KUKA KRL program: f1_Kuka_APT220T02S20.SRC

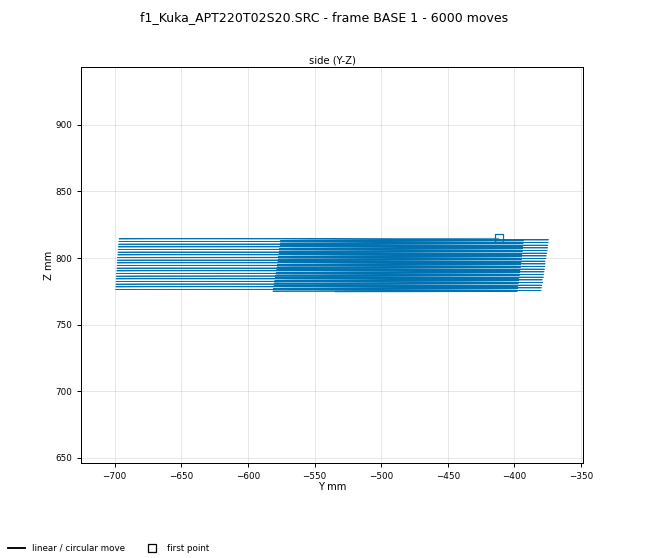
[picture p0: tool path of f1_Kuka_APT220T02S20.SRC in frame BASE 1, 6000 of 6001 moves have a stored position in this frame; points joined in program order, loops and branches not executed]
&ACCESS RVP
&REL 2
&PARAM TEMPLATE = C:\KRC\Roboter\Template\vorgabe
&PARAM EDITMASK = *
DEF f1_Kuka_APT220T02S20()


;FOLD INI;%{PE}%V3.2.0,%MKUKATPBASIS,%CINIT,%VCOMMON,%P
  ;FOLD BAS INI;%{E}%V3.2.0,%MKUKATPBASIS,%CINIT,%VINIT,%P
    GLOBAL INTERRUPT DECL 3 WHEN $STOPMESS==TRUE DO IR_STOPM ( )
    INTERRUPT ON 3
    BAS (#INITMOV,0 )
  ;ENDFOLD (BAS INI)
  ;FOLD USER INI;%{E}%V3.2.0,%MKUKATPUSER,%CINIT,%VINIT,%P
    ;Make your modifications here
  ;ENDFOLD (USER INI)
;ENDFOLD (INI)


;*** Make Null PTP Move
  PTP $pos_act

;*** Auto Load The Correct TOOL Data
  $tool=tool_data[2]

;*** Auto Load The Correct BASE Data
  $base=base_data[1]

  $ADVANCE = 5

;*** Restate Last Velocity
MMPM(30000.0)
SetRPM(8000)
LIN {X 0.104,Y -411.815,Z 814.863,A 0.000,B 0.000,C 90.000,E1 11.243} C_DIS
LIN {X -0.028,Y -415.979,Z 814.849,A 0.000,B 0.000,C 90.000,E1 8.859} C_DIS
LIN {X -0.170,Y -419.674,Z 814.838,A 0.000,B 0.000,C 90.000,E1 6.834} C_DIS
LIN {X 0.068,Y -422.792,Z 814.828,A 0.000,B 0.000,C 90.000,E1 5.106} C_DIS
LIN {X 0.041,Y -427.269,Z 814.815,A 0.000,B 0.000,C 90.000,E1 2.751} C_DIS
LIN {X 0.164,Y -433.422,Z 814.799,A 0.000,B 0.000,C 90.000,E1 359.771} C_DIS
LIN {X -0.033,Y -438.556,Z 814.786,A 0.000,B 0.000,C 90.000,E1 357.478} C_DIS
LIN {X 0.129,Y -442.521,Z 814.777,A 0.000,B 0.000,C 90.000,E1 355.812} C_DIS
LIN {X 0.097,Y -447.330,Z 814.766,A 0.000,B 0.000,C 90.000,E1 353.856} C_DIS
LIN {X 0.027,Y -451.496,Z 814.757,A 0.000,B 0.000,C 90.000,E1 352.243} C_DIS
LIN {X -0.123,Y -454.846,Z 814.750,A 0.000,B 0.000,C 90.000,E1 350.971} C_DIS
LIN {X -0.144,Y -456.848,Z 814.746,A 0.000,B 0.000,C 90.000,E1 350.330} C_DIS
LIN {X 0.078,Y -458.176,Z 814.744,A 0.000,B 0.000,C 90.000,E1 349.982} C_DIS
LIN {X 0.076,Y -460.220,Z 814.742,A 0.000,B 0.000,C 90.000,E1 349.634} C_DIS
LIN {X 0.046,Y -461.513,Z 814.741,A 0.000,B 0.000,C 90.000,E1 349.398} C_DIS
LIN {X 0.102,Y -464.808,Z 814.739,A 0.000,B 0.000,C 90.000,E1 348.993} C_DIS
LIN {X -0.030,Y -469.453,Z 814.737,A 0.000,B 0.000,C 90.000,E1 348.578} C_DIS
LIN {X 0.114,Y -476.009,Z 814.734,A 0.000,B 0.000,C 90.000,E1 348.049} C_DIS
LIN {X 0.121,Y -489.154,Z 814.729,A 0.000,B 0.000,C 90.000,E1 347.173} C_DIS
LIN {X -0.029,Y -500.125,Z 814.725,A 0.000,B 0.000,C 90.000,E1 346.464} C_DIS
LIN {X 0.244,Y -511.204,Z 814.721,A 0.000,B 0.000,C 90.000,E1 345.700} C_DIS
LIN {X 0.051,Y -523.694,Z 814.716,A 0.000,B 0.000,C 90.000,E1 344.866} C_DIS
LIN {X 0.230,Y -535.945,Z 814.711,A 0.000,B 0.000,C 90.000,E1 343.976} C_DIS
LIN {X 0.109,Y -546.247,Z 814.707,A 0.000,B 0.000,C 90.000,E1 343.196} C_DIS
LIN {X 0.238,Y -553.395,Z 814.703,A 0.000,B 0.000,C 90.000,E1 342.598} C_DIS
LIN {X 0.128,Y -558.933,Z 814.701,A 0.000,B 0.000,C 90.000,E1 342.127} C_DIS
LIN {X 0.040,Y -565.603,Z 814.697,A 0.000,B 0.000,C 90.000,E1 341.511} C_DIS
LIN {X 0.103,Y -571.834,Z 814.694,A 0.000,B 0.000,C 90.000,E1 340.859} C_DIS
LIN {X 0.161,Y -576.778,Z 814.691,A 0.000,B 0.000,C 90.000,E1 340.315} C_DIS
LIN {X 0.095,Y -582.280,Z 814.687,A 0.000,B 0.000,C 90.000,E1 339.645} C_DIS
LIN {X -0.127,Y -585.378,Z 814.685,A 0.000,B 0.000,C 90.000,E1 339.263} C_DIS
LIN {X 0.313,Y -591.974,Z 814.680,A 0.000,B 0.000,C 90.000,E1 338.284} C_DIS
LIN {X -0.223,Y -597.103,Z 814.675,A 0.000,B 0.000,C 90.000,E1 337.539} C_DIS
LIN {X -0.236,Y -603.578,Z 814.669,A 0.000,B 0.000,C 90.000,E1 336.485} C_DIS
LIN {X 0.161,Y -607.408,Z 814.666,A 0.000,B 0.000,C 90.000,E1 335.793} C_DIS
LIN {X -0.289,Y -614.208,Z 814.659,A 0.000,B 0.000,C 90.000,E1 334.665} C_DIS
LIN {X 0.202,Y -617.825,Z 814.656,A 0.000,B 0.000,C 90.000,E1 333.973} C_DIS
LIN {X 0.166,Y -624.634,Z 814.648,A 0.000,B 0.000,C 90.000,E1 332.692} C_DIS
LIN {X -0.052,Y -629.035,Z 814.643,A 0.000,B 0.000,C 90.000,E1 331.820} C_DIS
LIN {X 0.073,Y -634.391,Z 814.637,A 0.000,B 0.000,C 90.000,E1 330.667} C_DIS
LIN {X 0.046,Y -640.111,Z 814.630,A 0.000,B 0.000,C 90.000,E1 329.410} C_DIS
LIN {X 0.048,Y -644.293,Z 814.625,A 0.000,B 0.000,C 90.000,E1 328.408} C_DIS
LIN {X -0.026,Y -649.093,Z 814.618,A 0.000,B 0.000,C 90.000,E1 327.168} C_DIS
LIN {X 0.087,Y -652.631,Z 814.612,A 0.000,B 0.000,C 90.000,E1 326.167} C_DIS
LIN {X 0.063,Y -655.871,Z 814.607,A 0.000,B 0.000,C 90.000,E1 325.182} C_DIS
LIN {X 0.086,Y -658.937,Z 814.601,A 0.000,B 0.000,C 90.000,E1 324.196} C_DIS
LIN {X 0.103,Y -662.514,Z 814.594,A 0.000,B 0.000,C 90.000,E1 322.970} C_DIS
LIN {X 0.181,Y -665.628,Z 814.588,A 0.000,B 0.000,C 90.000,E1 321.743} C_DIS
LIN {X -0.215,Y -668.498,Z 814.581,A 0.000,B 0.000,C 90.000,E1 320.561} C_DIS
LIN {X 0.375,Y -671.116,Z 814.574,A 0.000,B 0.000,C 90.000,E1 319.299} C_DIS
LIN {X 0.046,Y -673.535,Z 814.567,A 0.000,B 0.000,C 90.000,E1 318.119} C_DIS
LIN {X 0.104,Y -674.880,Z 814.563,A 0.000,B 0.000,C 90.000,E1 317.391} C_DIS
LIN {X -0.220,Y -676.865,Z 814.557,A 0.000,B 0.000,C 90.000,E1 316.215} C_DIS
LIN {X -0.118,Y -677.962,Z 814.553,A 0.000,B 0.000,C 90.000,E1 315.486} C_DIS
LIN {X -0.003,Y -678.964,Z 814.549,A 0.000,B 0.000,C 90.000,E1 314.757} C_DIS
LIN {X 0.207,Y -680.520,Z 814.542,A 0.000,B 0.000,C 90.000,E1 313.542} C_DIS
LIN {X -0.397,Y -682.522,Z 814.533,A 0.000,B 0.000,C 90.000,E1 311.919} C_DIS
LIN {X -0.093,Y -683.878,Z 814.526,A 0.000,B 0.000,C 90.000,E1 310.701} C_DIS
LIN {X -0.161,Y -685.334,Z 814.518,A 0.000,B 0.000,C 90.000,E1 309.277} C_DIS
LIN {X -0.256,Y -686.461,Z 814.512,A 0.000,B 0.000,C 90.000,E1 308.096} C_DIS
LIN {X -0.130,Y -687.930,Z 814.502,A 0.000,B 0.000,C 90.000,E1 306.423} C_DIS
LIN {X -0.057,Y -688.887,Z 814.496,A 0.000,B 0.000,C 90.000,E1 305.231} C_DIS
LIN {X 0.031,Y -689.765,Z 814.489,A 0.000,B 0.000,C 90.000,E1 304.040} C_DIS
LIN {X -0.394,Y -690.938,Z 814.480,A 0.000,B 0.000,C 90.000,E1 302.418} C_DIS
LIN {X 0.163,Y -692.232,Z 814.471,A 0.000,B 0.000,C 90.000,E1 300.718} C_DIS
LIN {X 0.154,Y -693.018,Z 814.464,A 0.000,B 0.000,C 90.000,E1 299.539} C_DIS
LIN {X 0.048,Y -694.134,Z 814.455,A 0.000,B 0.000,C 90.000,E1 297.897} C_DIS
LIN {X 0.255,Y -695.322,Z 814.446,A 0.000,B 0.000,C 90.000,E1 296.232} C_DIS
LIN {X -0.064,Y -696.432,Z 814.438,A 0.000,B 0.000,C 90.000,E1 294.847} C_DIS
LIN {X -0.184,Y -696.729,Z 814.435,A 0.000,B 0.000,C 90.000,E1 294.387} C_DIS
LIN {X 0.044,Y -696.654,Z 814.433,A 0.000,B 0.000,C 90.000,E1 293.898} C_DIS
LIN {X 0.301,Y -696.552,Z 814.432,A 0.000,B 0.000,C 90.000,E1 293.643} C_DIS
LIN {X -0.083,Y -696.012,Z 814.430,A 0.000,B 0.000,C 90.000,E1 293.439} C_DIS
LIN {X 0.146,Y -694.455,Z 814.428,A 0.000,B 0.000,C 90.000,E1 292.950} C_DIS
LIN {X 0.269,Y -693.767,Z 814.427,A 0.000,B 0.000,C 90.000,E1 292.823} C_DIS
LIN {X 0.124,Y -692.737,Z 814.426,A 0.000,B 0.000,C 90.000,E1 292.717} C_DIS
LIN {X -0.273,Y -690.283,Z 814.425,A 0.000,B 0.000,C 90.000,E1 292.514} C_DIS
LIN {X -0.230,Y -687.459,Z 814.424,A 0.000,B 0.000,C 90.000,E1 292.280} C_DIS
LIN {X 0.023,Y -685.623,Z 814.423,A 0.000,B 0.000,C 90.000,E1 292.153} C_DIS
LIN {X 0.071,Y -681.364,Z 814.422,A 0.000,B 0.000,C 90.000,E1 291.972} C_DIS
LIN {X 0.256,Y -675.989,Z 814.421,A 0.000,B 0.000,C 90.000,E1 291.770} C_DIS
LIN {X 0.101,Y -671.875,Z 814.420,A 0.000,B 0.000,C 90.000,E1 291.663} C_DIS
LIN {X -0.284,Y -662.431,Z 814.420,A 0.000,B 0.000,C 90.000,E1 291.535} C_DIS
LIN {X 0.072,Y -648.303,Z 814.418,A 0.000,B 0.000,C 90.000,E1 291.280} C_DIS
LIN {X -0.110,Y -631.092,Z 814.417,A 0.000,B 0.000,C 90.000,E1 290.972} C_DIS
LIN {X 0.022,Y -621.065,Z 814.415,A 0.000,B 0.000,C 90.000,E1 290.737} C_DIS
LIN {X 0.190,Y -615.091,Z 814.414,A 0.000,B 0.000,C 90.000,E1 290.556} C_DIS
LIN {X 0.141,Y -607.421,Z 814.413,A 0.000,B 0.000,C 90.000,E1 290.301} C_DIS
LIN {X 0.257,Y -601.308,Z 814.411,A 0.000,B 0.000,C 90.000,E1 289.993} C_DIS
LIN {X -0.128,Y -600.257,Z 814.411,A 0.000,B 0.000,C 90.000,E1 289.939} C_DIS
LIN {X -0.126,Y -598.912,Z 814.410,A 0.000,B 0.000,C 90.000,E1 289.812} C_DIS
LIN {X 0.170,Y -597.816,Z 814.410,A 0.000,B 0.000,C 90.000,E1 289.704} C_DIS
LIN {X 0.129,Y -597.786,Z 814.410,A 0.000,B 0.000,C 90.000,E1 289.704} C_DIS
LIN {X 0.187,Y -597.270,Z 814.409,A 0.000,B 0.000,C 90.000,E1 289.523} C_DIS
LIN {X -0.213,Y -599.082,Z 814.406,A 0.000,B 0.000,C 90.000,E1 289.033} C_DIS
LIN {X 0.184,Y -600.898,Z 814.404,A 0.000,B 0.000,C 90.000,E1 288.671} C_DIS
LIN {X -0.033,Y -608.136,Z 814.397,A 0.000,B 0.000,C 90.000,E1 287.511} C_DIS
LIN {X -0.016,Y -611.361,Z 814.394,A 0.000,B 0.000,C 90.000,E1 286.858} C_DIS
LIN {X -0.006,Y -614.505,Z 814.389,A 0.000,B 0.000,C 90.000,E1 286.079} C_DIS
LIN {X 0.103,Y -616.101,Z 814.386,A 0.000,B 0.000,C 90.000,E1 285.552} C_DIS
LIN {X 0.158,Y -618.201,Z 814.382,A 0.000,B 0.000,C 90.000,E1 284.773} C_DIS
LIN {X -0.301,Y -619.069,Z 814.379,A 0.000,B 0.000,C 90.000,E1 284.300} C_DIS
LIN {X -0.151,Y -619.679,Z 814.376,A 0.000,B 0.000,C 90.000,E1 283.772} C_DIS
LIN {X -0.216,Y -620.183,Z 814.372,A 0.000,B 0.000,C 90.000,E1 283.008} C_DIS
LIN {X -0.054,Y -619.815,Z 814.369,A 0.000,B 0.000,C 90.000,E1 282.479} C_DIS
LIN {X 0.107,Y -619.178,Z 814.367,A 0.000,B 0.000,C 90.000,E1 281.951} C_DIS
LIN {X -0.117,Y -618.798,Z 814.365,A 0.000,B 0.000,C 90.000,E1 281.715} C_DIS
LIN {X 0.034,Y -617.514,Z 814.362,A 0.000,B 0.000,C 90.000,E1 281.186} C_DIS
LIN {X 0.174,Y -615.954,Z 814.359,A 0.000,B 0.000,C 90.000,E1 280.658} C_DIS
LIN {X 0.192,Y -613.967,Z 814.357,A 0.000,B 0.000,C 90.000,E1 280.141} C_DIS
LIN {X 0.129,Y -610.908,Z 814.353,A 0.000,B 0.000,C 90.000,E1 279.500} C_DIS
LIN {X 0.035,Y -607.088,Z 814.349,A 0.000,B 0.000,C 90.000,E1 278.859} C_DIS
LIN {X 0.001,Y -603.351,Z 814.346,A 0.000,B 0.000,C 90.000,E1 278.341} C_DIS
LIN {X 0.058,Y -598.365,Z 814.344,A 0.000,B 0.000,C 90.000,E1 277.814} C_DIS
LIN {X -0.103,Y -596.972,Z 814.343,A 0.000,B 0.000,C 90.000,E1 277.701} C_DIS
LIN {X -0.039,Y -590.807,Z 814.340,A 0.000,B 0.000,C 90.000,E1 277.239} C_DIS
LIN {X 0.031,Y -589.099,Z 814.340,A 0.000,B 0.000,C 90.000,E1 277.125} C_DIS
LIN {X 0.052,Y -581.500,Z 814.338,A 0.000,B 0.000,C 90.000,E1 276.777} C_DIS
LIN {X 0.185,Y -576.056,Z 814.337,A 0.000,B 0.000,C 90.000,E1 276.549} C_DIS
LIN {X 0.150,Y -571.955,Z 814.336,A 0.000,B 0.000,C 90.000,E1 276.429} C_DIS
LIN {X -0.190,Y -568.676,Z 814.335,A 0.000,B 0.000,C 90.000,E1 276.372} C_DIS
LIN {X 0.087,Y -566.129,Z 814.335,A 0.000,B 0.000,C 90.000,E1 276.315} C_DIS
LIN {X -0.135,Y -561.095,Z 814.335,A 0.000,B 0.000,C 90.000,E1 276.315} C_DIS
LIN {X -0.177,Y -554.630,Z 814.335,A 0.000,B 0.000,C 90.000,E1 276.315} C_DIS
LIN {X -0.087,Y -551.973,Z 814.335,A 0.000,B 0.000,C 90.000,E1 276.258} C_DIS
LIN {X -0.128,Y -551.928,Z 814.335,A 0.000,B 0.000,C 90.000,E1 276.258} C_DIS
LIN {X -0.079,Y -551.150,Z 814.334,A 0.000,B 0.000,C 90.000,E1 276.087} C_DIS
LIN {X 0.066,Y -550.419,Z 814.333,A 0.000,B 0.000,C 90.000,E1 275.967} C_DIS
LIN {X 0.023,Y -550.406,Z 814.333,A 0.000,B 0.000,C 90.000,E1 275.967} C_DIS
LIN {X -0.086,Y -549.667,Z 814.328,A 0.000,B 0.000,C 90.000,E1 275.106} C_DIS
LIN {X -0.271,Y -548.668,Z 814.319,A 0.000,B 0.000,C 90.000,E1 273.440} C_DIS
LIN {X 0.061,Y -547.489,Z 814.310,A 0.000,B 0.000,C 90.000,E1 271.718} C_DIS
LIN {X -0.260,Y -546.522,Z 814.302,A 0.000,B 0.000,C 90.000,E1 270.344} C_DIS
LIN {X 0.028,Y -545.133,Z 814.291,A 0.000,B 0.000,C 90.000,E1 268.339} C_DIS
LIN {X -0.231,Y -543.811,Z 814.280,A 0.000,B 0.000,C 90.000,E1 266.388} C_DIS
LIN {X -0.004,Y -542.786,Z 814.270,A 0.000,B 0.000,C 90.000,E1 264.666} C_DIS
LIN {X 0.152,Y -542.202,Z 814.266,A 0.000,B 0.000,C 90.000,E1 263.799} C_DIS
LIN {X -0.152,Y -540.991,Z 814.258,A 0.000,B 0.000,C 90.000,E1 262.413} C_DIS
LIN {X 0.121,Y -539.561,Z 814.248,A 0.000,B 0.000,C 90.000,E1 260.679} C_DIS
LIN {X -0.159,Y -538.124,Z 814.240,A 0.000,B 0.000,C 90.000,E1 259.285} C_DIS
LIN {X 0.160,Y -536.743,Z 814.232,A 0.000,B 0.000,C 90.000,E1 257.825} C_DIS
LIN {X 0.100,Y -534.985,Z 814.223,A 0.000,B 0.000,C 90.000,E1 256.117} C_DIS
LIN {X 0.140,Y -533.030,Z 814.213,A 0.000,B 0.000,C 90.000,E1 254.393} C_DIS
LIN {X 0.133,Y -531.035,Z 814.204,A 0.000,B 0.000,C 90.000,E1 252.670} C_DIS
LIN {X 0.215,Y -529.295,Z 814.196,A 0.000,B 0.000,C 90.000,E1 251.221} C_DIS
LIN {X -0.052,Y -527.408,Z 814.188,A 0.000,B 0.000,C 90.000,E1 249.806} C_DIS
LIN {X -0.023,Y -525.810,Z 814.181,A 0.000,B 0.000,C 90.000,E1 248.646} C_DIS
LIN {X -0.182,Y -523.314,Z 814.172,A 0.000,B 0.000,C 90.000,E1 246.922} C_DIS
LIN {X 0.017,Y -520.665,Z 814.162,A 0.000,B 0.000,C 90.000,E1 245.153} C_DIS
LIN {X -0.017,Y -519.255,Z 814.157,A 0.000,B 0.000,C 90.000,E1 244.280} C_DIS
LIN {X -0.028,Y -515.768,Z 814.146,A 0.000,B 0.000,C 90.000,E1 242.231} C_DIS
LIN {X 0.102,Y -513.047,Z 814.138,A 0.000,B 0.000,C 90.000,E1 240.745} C_DIS
LIN {X -0.117,Y -509.773,Z 814.128,A 0.000,B 0.000,C 90.000,E1 238.997} C_DIS
LIN {X 0.083,Y -507.346,Z 814.121,A 0.000,B 0.000,C 90.000,E1 237.788} C_DIS
LIN {X -0.183,Y -504.881,Z 814.115,A 0.000,B 0.000,C 90.000,E1 236.628} C_DIS
LIN {X 0.098,Y -501.636,Z 814.106,A 0.000,B 0.000,C 90.000,E1 235.102} C_DIS
LIN {X 0.153,Y -499.612,Z 814.101,A 0.000,B 0.000,C 90.000,E1 234.196} C_DIS
LIN {X 0.049,Y -496.682,Z 814.095,A 0.000,B 0.000,C 90.000,E1 233.004} C_DIS
LIN {X 0.051,Y -492.986,Z 814.086,A 0.000,B 0.000,C 90.000,E1 231.492} C_DIS
LIN {X -0.090,Y -490.767,Z 814.081,A 0.000,B 0.000,C 90.000,E1 230.598} C_DIS
LIN {X -0.150,Y -485.122,Z 814.068,A 0.000,B 0.000,C 90.000,E1 228.162} C_DIS
LIN {X 0.149,Y -480.300,Z 814.056,A 0.000,B 0.000,C 90.000,E1 225.972} C_DIS
LIN {X 0.193,Y -476.249,Z 814.045,A 0.000,B 0.000,C 90.000,E1 224.109} C_DIS
LIN {X 0.252,Y -471.518,Z 814.033,A 0.000,B 0.000,C 90.000,E1 221.919} C_DIS
LIN {X 0.034,Y -468.212,Z 814.024,A 0.000,B 0.000,C 90.000,E1 220.378} C_DIS
LIN {X 0.220,Y -464.338,Z 814.014,A 0.000,B 0.000,C 90.000,E1 218.463} C_DIS
LIN {X -0.224,Y -459.691,Z 814.002,A 0.000,B 0.000,C 90.000,E1 216.297} C_DIS
LIN {X 0.216,Y -455.724,Z 813.991,A 0.000,B 0.000,C 90.000,E1 214.326} C_DIS
LIN {X 0.144,Y -451.121,Z 813.978,A 0.000,B 0.000,C 90.000,E1 212.084} C_DIS
LIN {X -0.211,Y -445.800,Z 813.964,A 0.000,B 0.000,C 90.000,E1 209.539} C_DIS
LIN {X -0.072,Y -441.978,Z 813.953,A 0.000,B 0.000,C 90.000,E1 207.564} C_DIS
LIN {X -0.073,Y -438.830,Z 813.944,A 0.000,B 0.000,C 90.000,E1 205.924} C_DIS
LIN {X 0.046,Y -436.201,Z 813.937,A 0.000,B 0.000,C 90.000,E1 204.591} C_DIS
LIN {X -0.016,Y -431.661,Z 813.924,A 0.000,B 0.000,C 90.000,E1 202.280} C_DIS
LIN {X 0.028,Y -427.124,Z 813.911,A 0.000,B 0.000,C 90.000,E1 199.939} C_DIS
LIN {X 0.212,Y -423.868,Z 813.901,A 0.000,B 0.000,C 90.000,E1 198.236} C_DIS
LIN {X 0.072,Y -420.624,Z 813.892,A 0.000,B 0.000,C 90.000,E1 196.567} C_DIS
LIN {X 0.033,Y -416.744,Z 813.881,A 0.000,B 0.000,C 90.000,E1 194.537} C_DIS
LIN {X 0.219,Y -412.236,Z 813.868,A 0.000,B 0.000,C 90.000,E1 192.119} C_DIS
LIN {X -0.021,Y -409.021,Z 813.858,A 0.000,B 0.000,C 90.000,E1 190.433} C_DIS
LIN {X 0.088,Y -405.781,Z 813.848,A 0.000,B 0.000,C 90.000,E1 188.690} C_DIS
LIN {X 0.063,Y -401.258,Z 813.835,A 0.000,B 0.000,C 90.000,E1 186.258} C_DIS
LIN {X -0.153,Y -397.614,Z 813.823,A 0.000,B 0.000,C 90.000,E1 184.188} C_DIS
LIN {X 0.187,Y -393.457,Z 813.807,A 0.000,B 0.000,C 90.000,E1 181.318} C_DIS
LIN {X -0.106,Y -391.578,Z 813.800,A 0.000,B 0.000,C 90.000,E1 179.943} C_DIS
LIN {X 0.191,Y -389.034,Z 813.788,A 0.000,B 0.000,C 90.000,E1 177.764} C_DIS
LIN {X -0.159,Y -387.424,Z 813.780,A 0.000,B 0.000,C 90.000,E1 176.388} C_DIS
LIN {X -0.121,Y -384.233,Z 813.764,A 0.000,B 0.000,C 90.000,E1 173.514} C_DIS
LIN {X -0.187,Y -382.353,Z 813.754,A 0.000,B 0.000,C 90.000,E1 171.724} C_DIS
LIN {X -0.148,Y -381.037,Z 813.746,A 0.000,B 0.000,C 90.000,E1 170.274} C_DIS
LIN {X 0.196,Y -379.069,Z 813.734,A 0.000,B 0.000,C 90.000,E1 168.049} C_DIS
LIN {X -0.005,Y -376.771,Z 813.718,A 0.000,B 0.000,C 90.000,E1 165.172} C_DIS
LIN {X 0.071,Y -374.838,Z 813.697,A 0.000,B 0.000,C 90.000,E1 161.511} C_DIS
LIN {X -0.015,Y -374.344,Z 813.689,A 0.000,B 0.000,C 90.000,E1 160.061} C_DIS
LIN {X -0.075,Y -374.588,Z 813.669,A 0.000,B 0.000,C 90.000,E1 156.410} C_DIS
LIN {X -0.121,Y -375.577,Z 813.659,A 0.000,B 0.000,C 90.000,E1 154.588} C_DIS
LIN {X -0.119,Y -376.874,Z 813.651,A 0.000,B 0.000,C 90.000,E1 153.127} C_DIS
LIN {X -0.060,Y -378.378,Z 813.645,A 0.000,B 0.000,C 90.000,E1 152.025} C_DIS
LIN {X 0.076,Y -379.023,Z 813.643,A 0.000,B 0.000,C 90.000,E1 151.641} C_DIS
LIN {X -0.120,Y -379.539,Z 813.641,A 0.000,B 0.000,C 90.000,E1 151.307} C_DIS
LIN {X -0.029,Y -381.869,Z 813.635,A 0.000,B 0.000,C 90.000,E1 150.205} C_DIS
LIN {X 0.128,Y -383.752,Z 813.630,A 0.000,B 0.000,C 90.000,E1 149.459} C_DIS
LIN {X 0.106,Y -386.076,Z 813.626,A 0.000,B 0.000,C 90.000,E1 148.742} C_DIS
LIN {X -0.025,Y -389.025,Z 813.622,A 0.000,B 0.000,C 90.000,E1 148.043} C_DIS
LIN {X -0.174,Y -391.952,Z 813.619,A 0.000,B 0.000,C 90.000,E1 147.454} C_DIS
LIN {X 0.126,Y -394.852,Z 813.616,A 0.000,B 0.000,C 90.000,E1 146.914} C_DIS
LIN {X -0.005,Y -396.163,Z 813.615,A 0.000,B 0.000,C 90.000,E1 146.755} C_DIS
LIN {X 0.072,Y -399.489,Z 813.612,A 0.000,B 0.000,C 90.000,E1 146.215} C_DIS
LIN {X -0.024,Y -405.998,Z 813.608,A 0.000,B 0.000,C 90.000,E1 145.388} C_DIS
LIN {X -0.062,Y -408.930,Z 813.606,A 0.000,B 0.000,C 90.000,E1 145.055} C_DIS
LIN {X 0.133,Y -417.288,Z 813.601,A 0.000,B 0.000,C 90.000,E1 144.196} C_DIS
LIN {X 0.054,Y -421.954,Z 813.599,A 0.000,B 0.000,C 90.000,E1 143.783} C_DIS
LIN {X -0.145,Y -425.152,Z 813.597,A 0.000,B 0.000,C 90.000,E1 143.543} C_DIS
LIN {X 0.075,Y -429.554,Z 813.595,A 0.000,B 0.000,C 90.000,E1 143.130} C_DIS
LIN {X 0.224,Y -439.470,Z 813.590,A 0.000,B 0.000,C 90.000,E1 142.190} C_DIS
LIN {X 0.080,Y -443.548,Z 813.588,A 0.000,B 0.000,C 90.000,E1 141.778} C_DIS
LIN {X -0.021,Y -447.861,Z 813.585,A 0.000,B 0.000,C 90.000,E1 141.331} C_DIS
LIN {X -0.087,Y -450.694,Z 813.584,A 0.000,B 0.000,C 90.000,E1 141.045} C_DIS
LIN {X 0.156,Y -458.462,Z 813.578,A 0.000,B 0.000,C 90.000,E1 140.070} C_DIS
LIN {X -0.082,Y -463.322,Z 813.575,A 0.000,B 0.000,C 90.000,E1 139.461} C_DIS
LIN {X 0.162,Y -471.227,Z 813.569,A 0.000,B 0.000,C 90.000,E1 138.324} C_DIS
LIN {X 0.015,Y -475.454,Z 813.565,A 0.000,B 0.000,C 90.000,E1 137.715} C_DIS
LIN {X -0.048,Y -480.089,Z 813.561,A 0.000,B 0.000,C 90.000,E1 136.944} C_DIS
LIN {X -0.285,Y -486.198,Z 813.555,A 0.000,B 0.000,C 90.000,E1 135.891} C_DIS
LIN {X 0.091,Y -490.250,Z 813.551,A 0.000,B 0.000,C 90.000,E1 135.081} C_DIS
LIN {X 0.025,Y -499.146,Z 813.541,A 0.000,B 0.000,C 90.000,E1 133.419} C_DIS
LIN {X -0.087,Y -505.667,Z 813.534,A 0.000,B 0.000,C 90.000,E1 132.081} C_DIS
LIN {X 0.026,Y -508.416,Z 813.530,A 0.000,B 0.000,C 90.000,E1 131.472} C_DIS
LIN {X -0.079,Y -513.177,Z 813.524,A 0.000,B 0.000,C 90.000,E1 130.297} C_DIS
LIN {X -0.040,Y -514.911,Z 813.521,A 0.000,B 0.000,C 90.000,E1 129.850} C_DIS
LIN {X -0.120,Y -515.946,Z 813.520,A 0.000,B 0.000,C 90.000,E1 129.564} C_DIS
LIN {X -0.193,Y -517.186,Z 813.518,A 0.000,B 0.000,C 90.000,E1 129.277} C_DIS
LIN {X 0.066,Y -518.180,Z 813.516,A 0.000,B 0.000,C 90.000,E1 128.955} C_DIS
LIN {X 0.001,Y -519.346,Z 813.515,A 0.000,B 0.000,C 90.000,E1 128.669} C_DIS
LIN {X 0.073,Y -520.840,Z 813.512,A 0.000,B 0.000,C 90.000,E1 128.222} C_DIS
LIN {X -0.167,Y -522.656,Z 813.510,A 0.000,B 0.000,C 90.000,E1 127.810} C_DIS
LIN {X -0.298,Y -525.669,Z 813.505,A 0.000,B 0.000,C 90.000,E1 126.950} C_DIS
LIN {X -0.054,Y -527.879,Z 813.502,A 0.000,B 0.000,C 90.000,E1 126.343} C_DIS
LIN {X 0.342,Y -528.720,Z 813.500,A 0.000,B 0.000,C 90.000,E1 126.011} C_DIS
LIN {X 0.009,Y -529.810,Z 813.499,A 0.000,B 0.000,C 90.000,E1 125.758} C_DIS
LIN {X -0.011,Y -530.751,Z 813.497,A 0.000,B 0.000,C 90.000,E1 125.471} C_DIS
LIN {X -0.057,Y -532.744,Z 813.492,A 0.000,B 0.000,C 90.000,E1 124.612} C_DIS
LIN {X -0.069,Y -533.152,Z 813.491,A 0.000,B 0.000,C 90.000,E1 124.326} C_DIS
LIN {X -0.234,Y -534.210,Z 813.488,A 0.000,B 0.000,C 90.000,E1 123.913} C_DIS
LIN {X 0.305,Y -535.286,Z 813.486,A 0.000,B 0.000,C 90.000,E1 123.499} C_DIS
LIN {X 0.007,Y -535.804,Z 813.485,A 0.000,B 0.000,C 90.000,E1 123.245} C_DIS
LIN {X -0.174,Y -538.407,Z 813.481,A 0.000,B 0.000,C 90.000,E1 122.546} C_DIS
LIN {X 0.011,Y -541.360,Z 813.476,A 0.000,B 0.000,C 90.000,E1 121.671} C_DIS
LIN {X -0.251,Y -543.243,Z 813.473,A 0.000,B 0.000,C 90.000,E1 121.131} C_DIS
LIN {X -0.016,Y -545.867,Z 813.468,A 0.000,B 0.000,C 90.000,E1 120.256} C_DIS
LIN {X -0.025,Y -548.283,Z 813.463,A 0.000,B 0.000,C 90.000,E1 119.411} C_DIS
LIN {X -0.004,Y -550.556,Z 813.459,A 0.000,B 0.000,C 90.000,E1 118.565} C_DIS
LIN {X 0.045,Y -552.625,Z 813.454,A 0.000,B 0.000,C 90.000,E1 117.719} C_DIS
LIN {X 0.112,Y -554.466,Z 813.449,A 0.000,B 0.000,C 90.000,E1 116.873} C_DIS
LIN {X -0.050,Y -556.041,Z 813.445,A 0.000,B 0.000,C 90.000,E1 116.052} C_DIS
LIN {X 0.046,Y -557.342,Z 813.440,A 0.000,B 0.000,C 90.000,E1 115.207} C_DIS
LIN {X 0.304,Y -559.554,Z 813.431,A 0.000,B 0.000,C 90.000,E1 113.515} C_DIS
LIN {X -0.232,Y -560.850,Z 813.425,A 0.000,B 0.000,C 90.000,E1 112.461} C_DIS
LIN {X -0.229,Y -561.886,Z 813.419,A 0.000,B 0.000,C 90.000,E1 111.354} C_DIS
LIN {X -0.211,Y -562.561,Z 813.412,A 0.000,B 0.000,C 90.000,E1 110.248} C_DIS
LIN {X 0.024,Y -562.928,Z 813.408,A 0.000,B 0.000,C 90.000,E1 109.396} C_DIS
LIN {X 0.182,Y -563.292,Z 813.400,A 0.000,B 0.000,C 90.000,E1 108.000} C_DIS
LIN {X 0.093,Y -563.796,Z 813.389,A 0.000,B 0.000,C 90.000,E1 106.079} C_DIS
LIN {X 0.012,Y -564.785,Z 813.377,A 0.000,B 0.000,C 90.000,E1 103.883} C_DIS
LIN {X -0.302,Y -566.142,Z 813.365,A 0.000,B 0.000,C 90.000,E1 101.715} C_DIS
LIN {X 0.180,Y -567.330,Z 813.356,A 0.000,B 0.000,C 90.000,E1 100.018} C_DIS
LIN {X -0.067,Y -568.542,Z 813.347,A 0.000,B 0.000,C 90.000,E1 98.398} C_DIS
LIN {X -0.002,Y -569.297,Z 813.341,A 0.000,B 0.000,C 90.000,E1 97.296} C_DIS
LIN {X -0.106,Y -570.373,Z 813.330,A 0.000,B 0.000,C 90.000,E1 95.391} C_DIS
LIN {X 0.027,Y -571.050,Z 813.322,A 0.000,B 0.000,C 90.000,E1 94.012} C_DIS
LIN {X 0.136,Y -571.594,Z 813.315,A 0.000,B 0.000,C 90.000,E1 92.636} C_DIS
LIN {X 0.258,Y -572.132,Z 813.307,A 0.000,B 0.000,C 90.000,E1 91.260} C_DIS
LIN {X -0.055,Y -572.652,Z 813.298,A 0.000,B 0.000,C 90.000,E1 89.656} C_DIS
LIN {X 0.229,Y -573.082,Z 813.289,A 0.000,B 0.000,C 90.000,E1 87.993} C_DIS
LIN {X -0.052,Y -573.444,Z 813.280,A 0.000,B 0.000,C 90.000,E1 86.388} C_DIS
LIN {X -0.111,Y -573.897,Z 813.269,A 0.000,B 0.000,C 90.000,E1 84.489} C_DIS
LIN {X -0.040,Y -574.099,Z 813.263,A 0.000,B 0.000,C 90.000,E1 83.394} C_DIS
LIN {X -0.224,Y -574.426,Z 813.254,A 0.000,B 0.000,C 90.000,E1 81.781} C_DIS
LIN {X -0.237,Y -574.798,Z 813.245,A 0.000,B 0.000,C 90.000,E1 80.151} C_DIS
LIN {X 0.121,Y -575.153,Z 813.238,A 0.000,B 0.000,C 90.000,E1 78.757} C_DIS
LIN {X 0.027,Y -575.372,Z 813.230,A 0.000,B 0.000,C 90.000,E1 77.409} C_DIS
LIN {X -0.066,Y -575.464,Z 813.223,A 0.000,B 0.000,C 90.000,E1 76.061} C_DIS
LIN {X -0.026,Y -575.422,Z 813.215,A 0.000,B 0.000,C 90.000,E1 74.700} C_DIS
LIN {X 0.171,Y -575.372,Z 813.208,A 0.000,B 0.000,C 90.000,E1 73.323} C_DIS
LIN {X -0.183,Y -575.268,Z 813.203,A 0.000,B 0.000,C 90.000,E1 72.543} C_DIS
LIN {X -0.168,Y -574.996,Z 813.194,A 0.000,B 0.000,C 90.000,E1 70.913} C_DIS
LIN {X 0.031,Y -574.539,Z 813.185,A 0.000,B 0.000,C 90.000,E1 69.263} C_DIS
LIN {X -0.151,Y -574.120,Z 813.177,A 0.000,B 0.000,C 90.000,E1 67.922} C_DIS
LIN {X 0.092,Y -573.586,Z 813.170,A 0.000,B 0.000,C 90.000,E1 66.538} C_DIS
LIN {X -0.067,Y -572.830,Z 813.161,A 0.000,B 0.000,C 90.000,E1 64.921} C_DIS
LIN {X -0.111,Y -572.100,Z 813.153,A 0.000,B 0.000,C 90.000,E1 63.563} C_DIS
LIN {X -0.256,Y -571.282,Z 813.147,A 0.000,B 0.000,C 90.000,E1 62.487} C_DIS
LIN {X -0.050,Y -570.013,Z 813.139,A 0.000,B 0.000,C 90.000,E1 61.101} C_DIS
LIN {X 0.032,Y -568.796,Z 813.133,A 0.000,B 0.000,C 90.000,E1 59.999} C_DIS
LIN {X -0.111,Y -567.393,Z 813.127,A 0.000,B 0.000,C 90.000,E1 58.918} C_DIS
LIN {X 0.213,Y -565.762,Z 813.121,A 0.000,B 0.000,C 90.000,E1 57.788} C_DIS
LIN {X -0.079,Y -564.410,Z 813.117,A 0.000,B 0.000,C 90.000,E1 56.993} C_DIS
LIN {X 0.021,Y -562.314,Z 813.111,A 0.000,B 0.000,C 90.000,E1 55.881} C_DIS
LIN {X 0.093,Y -559.906,Z 813.104,A 0.000,B 0.000,C 90.000,E1 54.769} C_DIS
LIN {X 0.368,Y -557.891,Z 813.100,A 0.000,B 0.000,C 90.000,E1 53.909} C_DIS
LIN {X -0.238,Y -556.441,Z 813.097,A 0.000,B 0.000,C 90.000,E1 53.417} C_DIS
LIN {X 0.001,Y -554.003,Z 813.092,A 0.000,B 0.000,C 90.000,E1 52.557} C_DIS
LIN {X 0.210,Y -551.310,Z 813.087,A 0.000,B 0.000,C 90.000,E1 51.698} C_DIS
LIN {X -0.044,Y -548.206,Z 813.083,A 0.000,B 0.000,C 90.000,E1 50.884} C_DIS
LIN {X 0.051,Y -546.045,Z 813.080,A 0.000,B 0.000,C 90.000,E1 50.312} C_DIS
LIN {X -0.099,Y -543.063,Z 813.076,A 0.000,B 0.000,C 90.000,E1 49.622} C_DIS
LIN {X -0.273,Y -539.766,Z 813.072,A 0.000,B 0.000,C 90.000,E1 48.933} C_DIS
LIN {X 0.103,Y -536.861,Z 813.069,A 0.000,B 0.000,C 90.000,E1 48.324} C_DIS
LIN {X -0.125,Y -532.817,Z 813.065,A 0.000,B 0.000,C 90.000,E1 47.634} C_DIS
LIN {X -0.196,Y -529.291,Z 813.061,A 0.000,B 0.000,C 90.000,E1 47.067} C_DIS
LIN {X 0.261,Y -525.505,Z 813.058,A 0.000,B 0.000,C 90.000,E1 46.458} C_DIS
LIN {X 0.139,Y -521.189,Z 813.055,A 0.000,B 0.000,C 90.000,E1 45.891} C_DIS
LIN {X 0.042,Y -516.561,Z 813.052,A 0.000,B 0.000,C 90.000,E1 45.324} C_DIS
LIN {X 0.122,Y -511.762,Z 813.049,A 0.000,B 0.000,C 90.000,E1 44.757} C_DIS
LIN {X -0.151,Y -507.815,Z 813.046,A 0.000,B 0.000,C 90.000,E1 44.352} C_DIS
LIN {X -0.121,Y -502.158,Z 813.043,A 0.000,B 0.000,C 90.000,E1 43.785} C_DIS
LIN {X -0.005,Y -495.071,Z 813.039,A 0.000,B 0.000,C 90.000,E1 43.095} C_DIS
LIN {X 0.020,Y -490.496,Z 813.037,A 0.000,B 0.000,C 90.000,E1 42.690} C_DIS
LIN {X -0.092,Y -484.374,Z 813.034,A 0.000,B 0.000,C 90.000,E1 42.204} C_DIS
LIN {X 0.000,Y -476.617,Z 813.031,A 0.000,B 0.000,C 90.000,E1 41.595} C_DIS
LIN {X 0.008,Y -465.580,Z 813.027,A 0.000,B 0.000,C 90.000,E1 40.782} C_DIS
LIN {X 0.042,Y -447.997,Z 813.020,A 0.000,B 0.000,C 90.000,E1 39.519} C_DIS
LIN {X 0.186,Y -419.762,Z 813.008,A 0.000,B 0.000,C 90.000,E1 37.363} C_DIS
LIN {X -0.055,Y -409.184,Z 813.003,A 0.000,B 0.000,C 90.000,E1 36.503} C_DIS
LIN {X -0.154,Y -403.831,Z 813.000,A 0.000,B 0.000,C 90.000,E1 36.011} C_DIS
LIN {X 0.067,Y -400.406,Z 812.998,A 0.000,B 0.000,C 90.000,E1 35.598} C_DIS
LIN {X -0.069,Y -399.710,Z 812.997,A 0.000,B 0.000,C 90.000,E1 35.518} C_DIS
LIN {X -0.104,Y -399.686,Z 812.997,A 0.000,B 0.000,C 90.000,E1 35.518} C_DIS
LIN {X 0.017,Y -393.926,Z 812.977,A 0.000,B 0.000,C 90.000,E1 31.926} C_DIS
LIN {X -0.119,Y -393.291,Z 812.975,A 0.000,B 0.000,C 90.000,E1 31.592} C_DIS
LIN {X 0.080,Y -393.307,Z 812.974,A 0.000,B 0.000,C 90.000,E1 31.209} C_DIS
LIN {X 0.200,Y -394.544,Z 812.958,A 0.000,B 0.000,C 90.000,E1 28.359} C_DIS
LIN {X -0.068,Y -395.952,Z 812.944,A 0.000,B 0.000,C 90.000,E1 25.924} C_DIS
LIN {X 0.115,Y -397.896,Z 812.928,A 0.000,B 0.000,C 90.000,E1 23.078} C_DIS
LIN {X 0.179,Y -399.845,Z 812.915,A 0.000,B 0.000,C 90.000,E1 20.610} C_DIS
LIN {X -0.084,Y -403.459,Z 812.895,A 0.000,B 0.000,C 90.000,E1 17.149} C_DIS
LIN {X 0.116,Y -408.723,Z 812.874,A 0.000,B 0.000,C 90.000,E1 13.300} C_DIS
LIN {X 0.026,Y -412.098,Z 812.863,A 0.000,B 0.000,C 90.000,E1 11.243} C_DIS
LIN {X -0.098,Y -416.262,Z 812.849,A 0.000,B 0.000,C 90.000,E1 8.859} C_DIS
LIN {X 0.182,Y -419.962,Z 812.838,A 0.000,B 0.000,C 90.000,E1 6.777} C_DIS
LIN {X -0.062,Y -422.467,Z 812.830,A 0.000,B 0.000,C 90.000,E1 5.454} C_DIS
LIN {X -0.010,Y -427.531,Z 812.815,A 0.000,B 0.000,C 90.000,E1 2.751} C_DIS
LIN {X -0.182,Y -434.380,Z 812.797,A 0.000,B 0.000,C 90.000,E1 359.484} C_DIS
LIN {X 0.078,Y -439.558,Z 812.784,A 0.000,B 0.000,C 90.000,E1 357.135} C_DIS
LIN {X -0.185,Y -443.516,Z 812.775,A 0.000,B 0.000,C 90.000,E1 355.527} C_DIS
LIN {X -0.203,Y -448.358,Z 812.764,A 0.000,B 0.000,C 90.000,E1 353.571} C_DIS
LIN {X 0.002,Y -453.328,Z 812.753,A 0.000,B 0.000,C 90.000,E1 351.602} C_DIS
LIN {X 0.113,Y -455.866,Z 812.748,A 0.000,B 0.000,C 90.000,E1 350.622} C_DIS
LIN {X 0.102,Y -457.973,Z 812.744,A 0.000,B 0.000,C 90.000,E1 349.982} C_DIS
LIN {X -0.124,Y -459.717,Z 812.743,A 0.000,B 0.000,C 90.000,E1 349.690} C_DIS
LIN {X 0.111,Y -461.307,Z 812.741,A 0.000,B 0.000,C 90.000,E1 349.342} C_DIS
LIN {X 0.196,Y -463.726,Z 812.739,A 0.000,B 0.000,C 90.000,E1 348.993} C_DIS
LIN {X -0.202,Y -470.894,Z 812.735,A 0.000,B 0.000,C 90.000,E1 348.342} C_DIS
LIN {X 0.048,Y -477.310,Z 812.732,A 0.000,B 0.000,C 90.000,E1 347.813} C_DIS
LIN {X 0.136,Y -491.917,Z 812.727,A 0.000,B 0.000,C 90.000,E1 346.825} C_DIS
LIN {X 0.294,Y -507.842,Z 812.721,A 0.000,B 0.000,C 90.000,E1 345.755} C_DIS
LIN {X 0.034,Y -520.375,Z 812.716,A 0.000,B 0.000,C 90.000,E1 344.936} C_DIS
LIN {X -0.267,Y -532.642,Z 812.712,A 0.000,B 0.000,C 90.000,E1 344.102} C_DIS
LIN {X 0.085,Y -538.648,Z 812.709,A 0.000,B 0.000,C 90.000,E1 343.630} C_DIS
LIN {X -0.056,Y -547.527,Z 812.705,A 0.000,B 0.000,C 90.000,E1 342.960} C_DIS
LIN {X 0.080,Y -556.067,Z 812.701,A 0.000,B 0.000,C 90.000,E1 342.236} C_DIS
LIN {X -0.121,Y -561.526,Z 812.699,A 0.000,B 0.000,C 90.000,E1 341.764} C_DIS
LIN {X 0.234,Y -566.844,Z 812.696,A 0.000,B 0.000,C 90.000,E1 341.221} C_DIS
LIN {X -0.196,Y -573.138,Z 812.692,A 0.000,B 0.000,C 90.000,E1 340.604} C_DIS
LIN {X -0.045,Y -576.755,Z 812.690,A 0.000,B 0.000,C 90.000,E1 340.188} C_DIS
LIN {X -0.034,Y -581.214,Z 812.687,A 0.000,B 0.000,C 90.000,E1 339.645} C_DIS
LIN {X 0.214,Y -585.329,Z 812.684,A 0.000,B 0.000,C 90.000,E1 339.082} C_DIS
LIN {X 0.106,Y -591.906,Z 812.679,A 0.000,B 0.000,C 90.000,E1 338.156} C_DIS
LIN {X 0.120,Y -597.090,Z 812.674,A 0.000,B 0.000,C 90.000,E1 337.358} C_DIS
LIN {X 0.144,Y -602.777,Z 812.669,A 0.000,B 0.000,C 90.000,E1 336.433} C_DIS
LIN {X -0.020,Y -606.670,Z 812.666,A 0.000,B 0.000,C 90.000,E1 335.793} C_DIS
LIN {X 0.333,Y -613.514,Z 812.659,A 0.000,B 0.000,C 90.000,E1 334.588} C_DIS
LIN {X -0.011,Y -617.866,Z 812.655,A 0.000,B 0.000,C 90.000,E1 333.845} C_DIS
LIN {X -0.048,Y -624.041,Z 812.648,A 0.000,B 0.000,C 90.000,E1 332.692} C_DIS
LIN {X 0.271,Y -627.906,Z 812.644,A 0.000,B 0.000,C 90.000,E1 331.897} C_DIS
LIN {X -0.143,Y -634.504,Z 812.636,A 0.000,B 0.000,C 90.000,E1 330.539} C_DIS
LIN {X -0.218,Y -639.085,Z 812.631,A 0.000,B 0.000,C 90.000,E1 329.537} C_DIS
LIN {X -0.230,Y -643.376,Z 812.625,A 0.000,B 0.000,C 90.000,E1 328.535} C_DIS
LIN {X -0.189,Y -647.340,Z 812.620,A 0.000,B 0.000,C 90.000,E1 327.533} C_DIS
LIN {X -0.215,Y -651.918,Z 812.613,A 0.000,B 0.000,C 90.000,E1 326.294} C_DIS
LIN {X 0.212,Y -654.439,Z 812.609,A 0.000,B 0.000,C 90.000,E1 325.515} C_DIS
LIN {X 0.306,Y -658.403,Z 812.602,A 0.000,B 0.000,C 90.000,E1 324.276} C_DIS
LIN {X 0.312,Y -662.037,Z 812.595,A 0.000,B 0.000,C 90.000,E1 323.050} C_DIS
LIN {X 0.382,Y -665.232,Z 812.588,A 0.000,B 0.000,C 90.000,E1 321.823} C_DIS
LIN {X -0.023,Y -668.185,Z 812.581,A 0.000,B 0.000,C 90.000,E1 320.642} C_DIS
LIN {X -0.385,Y -670.899,Z 812.575,A 0.000,B 0.000,C 90.000,E1 319.461} C_DIS
LIN {X -0.273,Y -673.386,Z 812.568,A 0.000,B 0.000,C 90.000,E1 318.243} C_DIS
LIN {X 0.286,Y -674.789,Z 812.564,A 0.000,B 0.000,C 90.000,E1 317.472} C_DIS
LIN {X -0.009,Y -677.204,Z 812.556,A 0.000,B 0.000,C 90.000,E1 316.053} C_DIS
LIN {X 0.136,Y -678.666,Z 812.551,A 0.000,B 0.000,C 90.000,E1 315.081} C_DIS
LIN {X 0.387,Y -680.575,Z 812.543,A 0.000,B 0.000,C 90.000,E1 313.623} C_DIS
LIN {X -0.166,Y -682.866,Z 812.532,A 0.000,B 0.000,C 90.000,E1 311.757} C_DIS
LIN {X 0.092,Y -684.000,Z 812.527,A 0.000,B 0.000,C 90.000,E1 310.782} C_DIS
LIN {X 0.076,Y -685.672,Z 812.517,A 0.000,B 0.000,C 90.000,E1 309.116} C_DIS
LIN {X -0.062,Y -686.565,Z 812.512,A 0.000,B 0.000,C 90.000,E1 308.177} C_DIS
LIN {X 0.071,Y -688.067,Z 812.503,A 0.000,B 0.000,C 90.000,E1 306.503} C_DIS
LIN {X 0.150,Y -689.027,Z 812.496,A 0.000,B 0.000,C 90.000,E1 305.311} C_DIS
LIN {X 0.245,Y -689.918,Z 812.490,A 0.000,B 0.000,C 90.000,E1 304.119} C_DIS
LIN {X 0.200,Y -691.098,Z 812.481,A 0.000,B 0.000,C 90.000,E1 302.467} C_DIS
LIN {X 0.037,Y -692.560,Z 812.470,A 0.000,B 0.000,C 90.000,E1 300.590} C_DIS
LIN {X -0.206,Y -693.190,Z 812.465,A 0.000,B 0.000,C 90.000,E1 299.667} C_DIS
LIN {X -0.063,Y -694.450,Z 812.454,A 0.000,B 0.000,C 90.000,E1 297.769} C_DIS
LIN {X -0.219,Y -695.807,Z 812.444,A 0.000,B 0.000,C 90.000,E1 295.899} C_DIS
LIN {X -0.162,Y -696.673,Z 812.437,A 0.000,B 0.000,C 90.000,E1 294.719} C_DIS
LIN {X 0.353,Y -696.910,Z 812.435,A 0.000,B 0.000,C 90.000,E1 294.207} C_DIS
LIN {X -0.052,Y -696.720,Z 812.432,A 0.000,B 0.000,C 90.000,E1 293.770} C_DIS
LIN {X 0.204,Y -696.394,Z 812.431,A 0.000,B 0.000,C 90.000,E1 293.515} C_DIS
LIN {X -0.202,Y -694.832,Z 812.428,A 0.000,B 0.000,C 90.000,E1 293.078} C_DIS
LIN {X 0.046,Y -693.631,Z 812.427,A 0.000,B 0.000,C 90.000,E1 292.823} C_DIS
LIN {X -0.099,Y -692.548,Z 812.426,A 0.000,B 0.000,C 90.000,E1 292.717} C_DIS
LIN {X 0.203,Y -689.855,Z 812.425,A 0.000,B 0.000,C 90.000,E1 292.461} C_DIS
LIN {X -0.258,Y -687.130,Z 812.424,A 0.000,B 0.000,C 90.000,E1 292.280} C_DIS
LIN {X -0.001,Y -685.218,Z 812.423,A 0.000,B 0.000,C 90.000,E1 292.153} C_DIS
LIN {X 0.117,Y -680.925,Z 812.422,A 0.000,B 0.000,C 90.000,E1 291.972} C_DIS
LIN {X 0.101,Y -677.177,Z 812.421,A 0.000,B 0.000,C 90.000,E1 291.844} C_DIS
LIN {X -0.234,Y -671.892,Z 812.421,A 0.000,B 0.000,C 90.000,E1 291.716} C_DIS
LIN {X 0.147,Y -663.230,Z 812.420,A 0.000,B 0.000,C 90.000,E1 291.535} C_DIS
LIN {X 0.136,Y -647.158,Z 812.418,A 0.000,B 0.000,C 90.000,E1 291.280} C_DIS
LIN {X -0.081,Y -629.847,Z 812.417,A 0.000,B 0.000,C 90.000,E1 290.972} C_DIS
LIN {X 0.054,Y -619.851,Z 812.415,A 0.000,B 0.000,C 90.000,E1 290.737} C_DIS
LIN {X -0.270,Y -612.156,Z 812.414,A 0.000,B 0.000,C 90.000,E1 290.556} C_DIS
LIN {X 0.067,Y -607.024,Z 812.413,A 0.000,B 0.000,C 90.000,E1 290.355} C_DIS
LIN {X 0.267,Y -604.800,Z 812.413,A 0.000,B 0.000,C 90.000,E1 290.248} C_DIS
LIN {X -0.258,Y -601.090,Z 812.412,A 0.000,B 0.000,C 90.000,E1 290.120} C_DIS
LIN {X 0.253,Y -599.099,Z 812.411,A 0.000,B 0.000,C 90.000,E1 289.993} C_DIS
LIN {X 0.277,Y -595.410,Z 812.410,A 0.000,B 0.000,C 90.000,E1 289.758} C_DIS
LIN {X 0.019,Y -594.312,Z 812.409,A 0.000,B 0.000,C 90.000,E1 289.685} C_DIS
LIN {X -0.170,Y -593.774,Z 812.409,A 0.000,B 0.000,C 90.000,E1 289.631} C_DIS
LIN {X 0.123,Y -594.474,Z 812.406,A 0.000,B 0.000,C 90.000,E1 289.141} C_DIS
LIN {X -0.213,Y -598.299,Z 812.403,A 0.000,B 0.000,C 90.000,E1 288.489} C_DIS
LIN {X -0.145,Y -603.316,Z 812.398,A 0.000,B 0.000,C 90.000,E1 287.692} C_DIS
LIN {X -0.169,Y -606.774,Z 812.395,A 0.000,B 0.000,C 90.000,E1 287.040} C_DIS
LIN {X -0.204,Y -610.336,Z 812.390,A 0.000,B 0.000,C 90.000,E1 286.260} C_DIS
LIN {X -0.211,Y -612.828,Z 812.386,A 0.000,B 0.000,C 90.000,E1 285.481} C_DIS
LIN {X -0.111,Y -614.180,Z 812.383,A 0.000,B 0.000,C 90.000,E1 284.954} C_DIS
LIN {X 0.002,Y -615.229,Z 812.380,A 0.000,B 0.000,C 90.000,E1 284.426} C_DIS
LIN {X -0.084,Y -615.665,Z 812.379,A 0.000,B 0.000,C 90.000,E1 284.175} C_DIS
LIN {X 0.040,Y -616.172,Z 812.376,A 0.000,B 0.000,C 90.000,E1 283.647} C_DIS
LIN {X 0.170,Y -616.386,Z 812.373,A 0.000,B 0.000,C 90.000,E1 283.119} C_DIS
LIN {X -0.064,Y -616.349,Z 812.372,A 0.000,B 0.000,C 90.000,E1 282.883} C_DIS
LIN {X 0.069,Y -615.843,Z 812.369,A 0.000,B 0.000,C 90.000,E1 282.355} C_DIS
LIN {X 0.198,Y -615.110,Z 812.366,A 0.000,B 0.000,C 90.000,E1 281.827} C_DIS
LIN {X 0.321,Y -613.816,Z 812.363,A 0.000,B 0.000,C 90.000,E1 281.299} C_DIS
LIN {X -0.283,Y -612.182,Z 812.360,A 0.000,B 0.000,C 90.000,E1 280.838} C_DIS
LIN {X 0.167,Y -609.068,Z 812.356,A 0.000,B 0.000,C 90.000,E1 280.018} C_DIS
LIN {X 0.142,Y -606.530,Z 812.353,A 0.000,B 0.000,C 90.000,E1 279.500} C_DIS
LIN {X 0.196,Y -603.171,Z 812.350,A 0.000,B 0.000,C 90.000,E1 278.973} C_DIS
LIN {X 0.133,Y -599.134,Z 812.347,A 0.000,B 0.000,C 90.000,E1 278.454} C_DIS
LIN {X -0.057,Y -598.012,Z 812.346,A 0.000,B 0.000,C 90.000,E1 278.341} C_DIS
LIN {X 0.146,Y -593.929,Z 812.344,A 0.000,B 0.000,C 90.000,E1 277.936} C_DIS
LIN {X 0.144,Y -592.524,Z 812.344,A 0.000,B 0.000,C 90.000,E1 277.814} C_DIS
LIN {X 0.125,Y -589.330,Z 812.342,A 0.000,B 0.000,C 90.000,E1 277.587} C_DIS
LIN {X 0.015,Y -584.299,Z 812.341,A 0.000,B 0.000,C 90.000,E1 277.296} C_DIS
LIN {X 0.237,Y -582.380,Z 812.340,A 0.000,B 0.000,C 90.000,E1 277.182} C_DIS
LIN {X -0.112,Y -576.696,Z 812.339,A 0.000,B 0.000,C 90.000,E1 277.004} C_DIS
LIN {X -0.156,Y -575.178,Z 812.339,A 0.000,B 0.000,C 90.000,E1 276.947} C_DIS
LIN {X 0.217,Y -568.978,Z 812.338,A 0.000,B 0.000,C 90.000,E1 276.720} C_DIS
LIN {X 0.060,Y -568.190,Z 812.337,A 0.000,B 0.000,C 90.000,E1 276.720} C_DIS
LIN {X 0.223,Y -557.994,Z 812.337,A 0.000,B 0.000,C 90.000,E1 276.663} C_DIS
LIN {X -0.012,Y -554.606,Z 812.337,A 0.000,B 0.000,C 90.000,E1 276.663} C_DIS
LIN {X 0.200,Y -553.063,Z 812.337,A 0.000,B 0.000,C 90.000,E1 276.606} C_DIS
LIN {X -0.038,Y -551.791,Z 812.336,A 0.000,B 0.000,C 90.000,E1 276.549} C_DIS
LIN {X -0.244,Y -550.713,Z 812.336,A 0.000,B 0.000,C 90.000,E1 276.429} C_DIS
LIN {X 0.013,Y -550.214,Z 812.334,A 0.000,B 0.000,C 90.000,E1 276.030} C_DIS
LIN {X -0.064,Y -549.099,Z 812.323,A 0.000,B 0.000,C 90.000,E1 274.073} C_DIS
LIN {X 0.194,Y -548.364,Z 812.316,A 0.000,B 0.000,C 90.000,E1 272.922} C_DIS
LIN {X -0.100,Y -547.373,Z 812.309,A 0.000,B 0.000,C 90.000,E1 271.547} C_DIS
LIN {X 0.125,Y -546.409,Z 812.301,A 0.000,B 0.000,C 90.000,E1 270.115} C_DIS
LIN {X -0.174,Y -545.247,Z 812.291,A 0.000,B 0.000,C 90.000,E1 268.453} C_DIS
LIN {X 0.143,Y -543.729,Z 812.279,A 0.000,B 0.000,C 90.000,E1 266.159} C_DIS
LIN {X -0.195,Y -542.881,Z 812.271,A 0.000,B 0.000,C 90.000,E1 264.780} C_DIS
LIN {X -0.024,Y -542.078,Z 812.265,A 0.000,B 0.000,C 90.000,E1 263.628} C_DIS
LIN {X 0.201,Y -540.861,Z 812.257,A 0.000,B 0.000,C 90.000,E1 262.186} C_DIS
LIN {X -0.125,Y -539.944,Z 812.250,A 0.000,B 0.000,C 90.000,E1 261.084} C_DIS
LIN {X 0.066,Y -538.876,Z 812.244,A 0.000,B 0.000,C 90.000,E1 259.926} C_DIS
LIN {X 0.000,Y -536.914,Z 812.233,A 0.000,B 0.000,C 90.000,E1 257.937} C_DIS
LIN {X -0.048,Y -535.151,Z 812.224,A 0.000,B 0.000,C 90.000,E1 256.228} C_DIS
LIN {X -0.139,Y -533.217,Z 812.214,A 0.000,B 0.000,C 90.000,E1 254.519} C_DIS
LIN {X 0.011,Y -531.208,Z 812.204,A 0.000,B 0.000,C 90.000,E1 252.779} C_DIS
LIN {X 0.105,Y -529.476,Z 812.196,A 0.000,B 0.000,C 90.000,E1 251.329} C_DIS
LIN {X -0.153,Y -527.250,Z 812.187,A 0.000,B 0.000,C 90.000,E1 249.625} C_DIS
LIN {X 0.045,Y -525.146,Z 812.179,A 0.000,B 0.000,C 90.000,E1 248.156} C_DIS
LIN {X 0.026,Y -523.538,Z 812.172,A 0.000,B 0.000,C 90.000,E1 246.997} C_DIS
LIN {X 0.219,Y -520.912,Z 812.163,A 0.000,B 0.000,C 90.000,E1 245.229} C_DIS
LIN {X -0.285,Y -519.518,Z 812.158,A 0.000,B 0.000,C 90.000,E1 244.409} C_DIS
LIN {X -0.287,Y -515.992,Z 812.146,A 0.000,B 0.000,C 90.000,E1 242.359} C_DIS
LIN {X 0.100,Y -513.330,Z 812.138,A 0.000,B 0.000,C 90.000,E1 240.845} C_DIS
LIN {X 0.079,Y -510.027,Z 812.128,A 0.000,B 0.000,C 90.000,E1 239.076} C_DIS
LIN {X -0.153,Y -507.604,Z 812.122,A 0.000,B 0.000,C 90.000,E1 237.916} C_DIS
LIN {X -0.097,Y -504.516,Z 812.113,A 0.000,B 0.000,C 90.000,E1 236.421} C_DIS
LIN {X 0.177,Y -501.253,Z 812.105,A 0.000,B 0.000,C 90.000,E1 234.895} C_DIS
LIN {X -0.058,Y -499.955,Z 812.102,A 0.000,B 0.000,C 90.000,E1 234.322} C_DIS
LIN {X -0.282,Y -496.226,Z 812.093,A 0.000,B 0.000,C 90.000,E1 232.844} C_DIS
LIN {X -0.137,Y -493.301,Z 812.087,A 0.000,B 0.000,C 90.000,E1 231.618} C_DIS
LIN {X 0.109,Y -489.562,Z 812.078,A 0.000,B 0.000,C 90.000,E1 230.070} C_DIS
LIN {X 0.197,Y -484.664,Z 812.066,A 0.000,B 0.000,C 90.000,E1 227.919} C_DIS
LIN {X -0.196,Y -479.894,Z 812.054,A 0.000,B 0.000,C 90.000,E1 225.810} C_DIS
LIN {X -0.271,Y -476.553,Z 812.046,A 0.000,B 0.000,C 90.000,E1 224.271} C_DIS
LIN {X -0.024,Y -470.477,Z 812.030,A 0.000,B 0.000,C 90.000,E1 221.434} C_DIS
LIN {X 0.273,Y -465.842,Z 812.018,A 0.000,B 0.000,C 90.000,E1 219.197} C_DIS
LIN {X 0.084,Y -464.612,Z 812.014,A 0.000,B 0.000,C 90.000,E1 218.588} C_DIS
LIN {X -0.246,Y -459.252,Z 812.000,A 0.000,B 0.000,C 90.000,E1 216.091} C_DIS
LIN {X -0.175,Y -455.970,Z 811.992,A 0.000,B 0.000,C 90.000,E1 214.485} C_DIS
LIN {X 0.013,Y -451.417,Z 811.979,A 0.000,B 0.000,C 90.000,E1 212.212} C_DIS
LIN {X 0.052,Y -446.072,Z 811.965,A 0.000,B 0.000,C 90.000,E1 209.617} C_DIS
LIN {X 0.202,Y -442.238,Z 811.954,A 0.000,B 0.000,C 90.000,E1 207.641} C_DIS
LIN {X -0.154,Y -438.471,Z 811.943,A 0.000,B 0.000,C 90.000,E1 205.720} C_DIS
LIN {X -0.059,Y -436.490,Z 811.937,A 0.000,B 0.000,C 90.000,E1 204.719} C_DIS
LIN {X 0.053,Y -431.980,Z 811.924,A 0.000,B 0.000,C 90.000,E1 202.386} C_DIS
LIN {X 0.140,Y -428.072,Z 811.913,A 0.000,B 0.000,C 90.000,E1 200.375} C_DIS
LIN {X -0.053,Y -424.887,Z 811.904,A 0.000,B 0.000,C 90.000,E1 198.725} C_DIS
LIN {X 0.132,Y -420.944,Z 811.893,A 0.000,B 0.000,C 90.000,E1 196.677} C_DIS
LIN {X -0.013,Y -417.077,Z 811.881,A 0.000,B 0.000,C 90.000,E1 194.662} C_DIS
LIN {X -0.174,Y -411.910,Z 811.866,A 0.000,B 0.000,C 90.000,E1 191.951} C_DIS
LIN {X 0.039,Y -409.377,Z 811.859,A 0.000,B 0.000,C 90.000,E1 190.546} C_DIS
LIN {X 0.165,Y -405.474,Z 811.847,A 0.000,B 0.000,C 90.000,E1 188.454} C_DIS
LIN {X 0.081,Y -400.990,Z 811.834,A 0.000,B 0.000,C 90.000,E1 186.030} C_DIS
LIN {X -0.080,Y -397.963,Z 811.824,A 0.000,B 0.000,C 90.000,E1 184.302} C_DIS
LIN {X -0.194,Y -393.289,Z 811.806,A 0.000,B 0.000,C 90.000,E1 181.146} C_DIS
LIN {X -0.020,Y -391.881,Z 811.800,A 0.000,B 0.000,C 90.000,E1 180.057} C_DIS
LIN {X 0.136,Y -390.603,Z 811.794,A 0.000,B 0.000,C 90.000,E1 178.969} C_DIS
LIN {X 0.034,Y -388.219,Z 811.783,A 0.000,B 0.000,C 90.000,E1 176.846} C_DIS
LIN {X -0.006,Y -384.610,Z 811.765,A 0.000,B 0.000,C 90.000,E1 173.628} C_DIS
LIN {X -0.062,Y -382.737,Z 811.755,A 0.000,B 0.000,C 90.000,E1 171.837} C_DIS
LIN {X -0.101,Y -381.041,Z 811.745,A 0.000,B 0.000,C 90.000,E1 170.038} C_DIS
LIN {X 0.152,Y -378.827,Z 811.731,A 0.000,B 0.000,C 90.000,E1 167.465} C_DIS
LIN {X 0.033,Y -376.650,Z 811.714,A 0.000,B 0.000,C 90.000,E1 164.574} C_DIS
LIN {X 0.129,Y -375.002,Z 811.696,A 0.000,B 0.000,C 90.000,E1 161.275} C_DIS
LIN {X -0.078,Y -374.567,Z 811.674,A 0.000,B 0.000,C 90.000,E1 157.283} C_DIS
LIN {X 0.091,Y -375.790,Z 811.658,A 0.000,B 0.000,C 90.000,E1 154.332} C_DIS
LIN {X 0.097,Y -377.086,Z 811.649,A 0.000,B 0.000,C 90.000,E1 152.871} C_DIS
LIN {X -0.037,Y -379.034,Z 811.641,A 0.000,B 0.000,C 90.000,E1 151.435} C_DIS
LIN {X 0.048,Y -381.023,Z 811.635,A 0.000,B 0.000,C 90.000,E1 150.333} C_DIS
LIN {X 0.005,Y -382.738,Z 811.631,A 0.000,B 0.000,C 90.000,E1 149.616} C_DIS
LIN {X -0.182,Y -385.449,Z 811.626,A 0.000,B 0.000,C 90.000,E1 148.742} C_DIS
LIN {X 0.011,Y -388.128,Z 811.622,A 0.000,B 0.000,C 90.000,E1 147.995} C_DIS
LIN {X -0.151,Y -389.749,Z 811.620,A 0.000,B 0.000,C 90.000,E1 147.661} C_DIS
LIN {X 0.231,Y -391.290,Z 811.618,A 0.000,B 0.000,C 90.000,E1 147.248} C_DIS
LIN {X 0.080,Y -393.177,Z 811.616,A 0.000,B 0.000,C 90.000,E1 146.914} C_DIS
LIN {X -0.065,Y -394.903,Z 811.614,A 0.000,B 0.000,C 90.000,E1 146.580} C_DIS
LIN {X 0.222,Y -397.837,Z 811.611,A 0.000,B 0.000,C 90.000,E1 146.008} C_DIS
LIN {X 0.087,Y -405.764,Z 811.606,A 0.000,B 0.000,C 90.000,E1 144.975} C_DIS
LIN {X 0.053,Y -412.655,Z 811.601,A 0.000,B 0.000,C 90.000,E1 144.149} C_DIS
LIN {X 0.124,Y -423.288,Z 811.595,A 0.000,B 0.000,C 90.000,E1 143.130} C_DIS
LIN {X 0.123,Y -426.286,Z 811.594,A 0.000,B 0.000,C 90.000,E1 142.844} C_DIS
LIN {X 0.041,Y -433.376,Z 811.590,A 0.000,B 0.000,C 90.000,E1 142.145} C_DIS
LIN {X 0.206,Y -436.418,Z 811.588,A 0.000,B 0.000,C 90.000,E1 141.823} C_DIS
LIN {X -0.148,Y -445.866,Z 811.582,A 0.000,B 0.000,C 90.000,E1 140.803} C_DIS
LIN {X 0.058,Y -455.224,Z 811.576,A 0.000,B 0.000,C 90.000,E1 139.666} C_DIS
LIN {X 0.173,Y -461.186,Z 811.572,A 0.000,B 0.000,C 90.000,E1 138.852} C_DIS
LIN {X -0.046,Y -465.665,Z 811.568,A 0.000,B 0.000,C 90.000,E1 138.243} C_DIS
LIN {X 0.044,Y -468.916,Z 811.565,A 0.000,B 0.000,C 90.000,E1 137.757} C_DIS
LIN {X -0.160,Y -472.017,Z 811.563,A 0.000,B 0.000,C 90.000,E1 137.310} C_DIS
LIN {X -0.154,Y -478.580,Z 811.557,A 0.000,B 0.000,C 90.000,E1 136.215} C_DIS
LIN {X 0.004,Y -485.488,Z 811.550,A 0.000,B 0.000,C 90.000,E1 134.960} C_DIS
LIN {X 0.031,Y -489.672,Z 811.546,A 0.000,B 0.000,C 90.000,E1 134.190} C_DIS
LIN {X 0.009,Y -496.279,Z 811.539,A 0.000,B 0.000,C 90.000,E1 132.975} C_DIS
LIN {X 0.045,Y -499.366,Z 811.535,A 0.000,B 0.000,C 90.000,E1 132.366} C_DIS
LIN {X 0.006,Y -501.400,Z 811.533,A 0.000,B 0.000,C 90.000,E1 131.919} C_DIS
LIN {X -0.032,Y -505.578,Z 811.528,A 0.000,B 0.000,C 90.000,E1 131.067} C_DIS
LIN {X -0.140,Y -508.594,Z 811.524,A 0.000,B 0.000,C 90.000,E1 130.334} C_DIS
LIN {X 0.088,Y -510.145,Z 811.522,A 0.000,B 0.000,C 90.000,E1 130.011} C_DIS
LIN {X 0.112,Y -512.019,Z 811.520,A 0.000,B 0.000,C 90.000,E1 129.564} C_DIS
LIN {X -0.056,Y -514.295,Z 811.517,A 0.000,B 0.000,C 90.000,E1 128.991} C_DIS
LIN {X -0.009,Y -516.366,Z 811.514,A 0.000,B 0.000,C 90.000,E1 128.543} C_DIS
LIN {X 0.049,Y -518.139,Z 811.512,A 0.000,B 0.000,C 90.000,E1 128.096} C_DIS
LIN {X 0.114,Y -519.837,Z 811.509,A 0.000,B 0.000,C 90.000,E1 127.649} C_DIS
LIN {X 0.058,Y -521.246,Z 811.508,A 0.000,B 0.000,C 90.000,E1 127.363} C_DIS
LIN {X -0.087,Y -524.522,Z 811.503,A 0.000,B 0.000,C 90.000,E1 126.503} C_DIS
LIN {X -0.301,Y -526.436,Z 811.500,A 0.000,B 0.000,C 90.000,E1 126.091} C_DIS
LIN {X 0.040,Y -529.443,Z 811.496,A 0.000,B 0.000,C 90.000,E1 125.185} C_DIS
LIN {X -0.003,Y -530.742,Z 811.492,A 0.000,B 0.000,C 90.000,E1 124.612} C_DIS
LIN {X -0.042,Y -531.467,Z 811.491,A 0.000,B 0.000,C 90.000,E1 124.405} C_DIS
LIN {X -0.229,Y -533.494,Z 811.487,A 0.000,B 0.000,C 90.000,E1 123.706} C_DIS
LIN {X 0.047,Y -536.182,Z 811.483,A 0.000,B 0.000,C 90.000,E1 122.959} C_DIS
LIN {X 0.207,Y -539.371,Z 811.478,A 0.000,B 0.000,C 90.000,E1 122.084} C_DIS
LIN {X -0.057,Y -542.334,Z 811.474,A 0.000,B 0.000,C 90.000,E1 121.258} C_DIS
LIN {X -0.108,Y -545.060,Z 811.469,A 0.000,B 0.000,C 90.000,E1 120.413} C_DIS
LIN {X -0.099,Y -548.326,Z 811.463,A 0.000,B 0.000,C 90.000,E1 119.283} C_DIS
LIN {X -0.077,Y -550.665,Z 811.458,A 0.000,B 0.000,C 90.000,E1 118.437} C_DIS
LIN {X -0.027,Y -552.751,Z 811.453,A 0.000,B 0.000,C 90.000,E1 117.590} C_DIS
LIN {X 0.265,Y -554.027,Z 811.450,A 0.000,B 0.000,C 90.000,E1 117.001} C_DIS
LIN {X 0.098,Y -555.687,Z 811.446,A 0.000,B 0.000,C 90.000,E1 116.181} C_DIS
LIN {X -0.093,Y -556.695,Z 811.442,A 0.000,B 0.000,C 90.000,E1 115.643} C_DIS
LIN {X 0.058,Y -558.250,Z 811.436,A 0.000,B 0.000,C 90.000,E1 114.515} C_DIS
LIN {X 0.027,Y -560.061,Z 811.429,A 0.000,B 0.000,C 90.000,E1 113.131} C_DIS
LIN {X -0.298,Y -561.004,Z 811.424,A 0.000,B 0.000,C 90.000,E1 112.333} C_DIS
LIN {X -0.295,Y -562.038,Z 811.418,A 0.000,B 0.000,C 90.000,E1 111.227} C_DIS
LIN {X 0.041,Y -562.843,Z 811.410,A 0.000,B 0.000,C 90.000,E1 109.812} C_DIS
LIN {X 0.193,Y -563.309,Z 811.402,A 0.000,B 0.000,C 90.000,E1 108.417} C_DIS
LIN {X -0.289,Y -563.937,Z 811.390,A 0.000,B 0.000,C 90.000,E1 106.260} C_DIS
LIN {X 0.186,Y -564.924,Z 811.378,A 0.000,B 0.000,C 90.000,E1 104.008} C_DIS
LIN {X 0.004,Y -566.299,Z 811.366,A 0.000,B 0.000,C 90.000,E1 101.827} C_DIS
LIN {X 0.001,Y -567.677,Z 811.355,A 0.000,B 0.000,C 90.000,E1 99.905} C_DIS
LIN {X -0.151,Y -568.891,Z 811.346,A 0.000,B 0.000,C 90.000,E1 98.276} C_DIS
LIN {X -0.160,Y -569.630,Z 811.340,A 0.000,B 0.000,C 90.000,E1 97.182} C_DIS
LIN {X -0.253,Y -570.704,Z 811.329,A 0.000,B 0.000,C 90.000,E1 95.277} C_DIS
LIN {X -0.113,Y -571.383,Z 811.322,A 0.000,B 0.000,C 90.000,E1 93.898} C_DIS
LIN {X 0.004,Y -571.930,Z 811.314,A 0.000,B 0.000,C 90.000,E1 92.522} C_DIS
LIN {X 0.271,Y -572.557,Z 811.305,A 0.000,B 0.000,C 90.000,E1 90.859} C_DIS
LIN {X -0.033,Y -573.077,Z 811.296,A 0.000,B 0.000,C 90.000,E1 89.255} C_DIS
LIN {X 0.258,Y -573.508,Z 811.287,A 0.000,B 0.000,C 90.000,E1 87.593} C_DIS
LIN {X -0.021,Y -573.839,Z 811.278,A 0.000,B 0.000,C 90.000,E1 85.988} C_DIS
LIN {X -0.213,Y -574.214,Z 811.269,A 0.000,B 0.000,C 90.000,E1 84.375} C_DIS
LIN {X -0.139,Y -574.431,Z 811.263,A 0.000,B 0.000,C 90.000,E1 83.280} C_DIS
LIN {X -0.237,Y -574.767,Z 811.254,A 0.000,B 0.000,C 90.000,E1 81.659} C_DIS
LIN {X 0.031,Y -575.068,Z 811.246,A 0.000,B 0.000,C 90.000,E1 80.274} C_DIS
LIN {X 0.140,Y -575.467,Z 811.237,A 0.000,B 0.000,C 90.000,E1 78.634} C_DIS
LIN {X 0.059,Y -575.644,Z 811.229,A 0.000,B 0.000,C 90.000,E1 77.285} C_DIS
LIN {X -0.023,Y -575.720,Z 811.222,A 0.000,B 0.000,C 90.000,E1 75.936} C_DIS
LIN {X 0.027,Y -575.637,Z 811.214,A 0.000,B 0.000,C 90.000,E1 74.574} C_DIS
LIN {X 0.234,Y -575.563,Z 811.207,A 0.000,B 0.000,C 90.000,E1 73.196} C_DIS
LIN {X 0.075,Y -575.385,Z 811.201,A 0.000,B 0.000,C 90.000,E1 72.127} C_DIS
LIN {X -0.092,Y -575.147,Z 811.193,A 0.000,B 0.000,C 90.000,E1 70.786} C_DIS
LIN {X 0.116,Y -574.662,Z 811.184,A 0.000,B 0.000,C 90.000,E1 69.135} C_DIS
LIN {X -0.063,Y -574.217,Z 811.177,A 0.000,B 0.000,C 90.000,E1 67.794} C_DIS
LIN {X -0.207,Y -573.547,Z 811.168,A 0.000,B 0.000,C 90.000,E1 66.177} C_DIS
LIN {X -0.135,Y -572.712,Z 811.159,A 0.000,B 0.000,C 90.000,E1 64.537} C_DIS
LIN {X -0.177,Y -571.898,Z 811.151,A 0.000,B 0.000,C 90.000,E1 63.179} C_DIS
LIN {X -0.161,Y -571.205,Z 811.146,A 0.000,B 0.000,C 90.000,E1 62.359} C_DIS
LIN {X 0.042,Y -569.865,Z 811.139,A 0.000,B 0.000,C 90.000,E1 60.973} C_DIS
LIN {X 0.298,Y -568.960,Z 811.134,A 0.000,B 0.000,C 90.000,E1 60.127} C_DIS
LIN {X 0.049,Y -567.913,Z 811.130,A 0.000,B 0.000,C 90.000,E1 59.331} C_DIS
LIN {X -0.212,Y -566.733,Z 811.125,A 0.000,B 0.000,C 90.000,E1 58.535} C_DIS
LIN {X 0.092,Y -564.996,Z 811.119,A 0.000,B 0.000,C 90.000,E1 57.406} C_DIS
LIN {X 0.096,Y -563.520,Z 811.114,A 0.000,B 0.000,C 90.000,E1 56.580} C_DIS
LIN {X 0.085,Y -561.876,Z 811.110,A 0.000,B 0.000,C 90.000,E1 55.754} C_DIS
LIN {X 0.377,Y -560.077,Z 811.105,A 0.000,B 0.000,C 90.000,E1 54.895} C_DIS
LIN {X -0.125,Y -558.040,Z 811.101,A 0.000,B 0.000,C 90.000,E1 54.116} C_DIS
LIN {X 0.134,Y -555.783,Z 811.096,A 0.000,B 0.000,C 90.000,E1 53.256} C_DIS
LIN {X 0.099,Y -552.311,Z 811.090,A 0.000,B 0.000,C 90.000,E1 52.145} C_DIS
LIN {X -0.205,Y -550.415,Z 811.087,A 0.000,B 0.000,C 90.000,E1 51.618} C_DIS
LIN {X 0.306,Y -547.239,Z 811.082,A 0.000,B 0.000,C 90.000,E1 50.723} C_DIS
LIN {X 0.013,Y -543.808,Z 811.077,A 0.000,B 0.000,C 90.000,E1 49.908} C_DIS
LIN {X 0.236,Y -541.904,Z 811.075,A 0.000,B 0.000,C 90.000,E1 49.461} C_DIS
LIN {X -0.133,Y -539.211,Z 811.072,A 0.000,B 0.000,C 90.000,E1 48.933} C_DIS
LIN {X 0.238,Y -536.286,Z 811.069,A 0.000,B 0.000,C 90.000,E1 48.324} C_DIS
LIN {X 0.003,Y -532.140,Z 811.065,A 0.000,B 0.000,C 90.000,E1 47.634} C_DIS
LIN {X -0.073,Y -528.535,Z 811.061,A 0.000,B 0.000,C 90.000,E1 47.067} C_DIS
LIN {X -0.012,Y -524.638,Z 811.058,A 0.000,B 0.000,C 90.000,E1 46.500} C_DIS
LIN {X 0.239,Y -520.244,Z 811.055,A 0.000,B 0.000,C 90.000,E1 45.891} C_DIS
LIN {X -0.059,Y -516.758,Z 811.053,A 0.000,B 0.000,C 90.000,E1 45.486} C_DIS
LIN {X 0.155,Y -510.550,Z 811.049,A 0.000,B 0.000,C 90.000,E1 44.757} C_DIS
LIN {X 0.001,Y -506.628,Z 811.046,A 0.000,B 0.000,C 90.000,E1 44.352} C_DIS
LIN {X 0.013,Y -499.613,Z 811.043,A 0.000,B 0.000,C 90.000,E1 43.662} C_DIS
LIN {X -0.089,Y -493.858,Z 811.040,A 0.000,B 0.000,C 90.000,E1 43.137} C_DIS
LIN {X 0.028,Y -487.815,Z 811.037,A 0.000,B 0.000,C 90.000,E1 42.609} C_DIS
LIN {X 0.156,Y -480.227,Z 811.034,A 0.000,B 0.000,C 90.000,E1 42.000} C_DIS
LIN {X 0.016,Y -470.688,Z 811.030,A 0.000,B 0.000,C 90.000,E1 41.310} C_DIS
LIN {X 0.036,Y -461.124,Z 811.026,A 0.000,B 0.000,C 90.000,E1 40.620} C_DIS
LIN {X 0.266,Y -446.770,Z 811.020,A 0.000,B 0.000,C 90.000,E1 39.564} C_DIS
LIN {X 0.080,Y -421.496,Z 811.009,A 0.000,B 0.000,C 90.000,E1 37.684} C_DIS
LIN {X 0.112,Y -409.351,Z 811.004,A 0.000,B 0.000,C 90.000,E1 36.664} C_DIS
LIN {X 0.074,Y -403.355,Z 811.001,A 0.000,B 0.000,C 90.000,E1 36.091} C_DIS
LIN {X 0.062,Y -400.142,Z 810.999,A 0.000,B 0.000,C 90.000,E1 35.724} C_DIS
LIN {X 0.033,Y -400.110,Z 810.999,A 0.000,B 0.000,C 90.000,E1 35.724} C_DIS
LIN {X 0.082,Y -393.606,Z 810.976,A 0.000,B 0.000,C 90.000,E1 31.720} C_DIS
LIN {X -0.190,Y -393.428,Z 810.976,A 0.000,B 0.000,C 90.000,E1 31.671} C_DIS
LIN {X 0.007,Y -394.529,Z 810.961,A 0.000,B 0.000,C 90.000,E1 28.899} C_DIS
LIN {X 0.100,Y -395.877,Z 810.947,A 0.000,B 0.000,C 90.000,E1 26.411} C_DIS
LIN {X 0.110,Y -397.745,Z 810.931,A 0.000,B 0.000,C 90.000,E1 23.590} C_DIS
LIN {X 0.030,Y -399.957,Z 810.916,A 0.000,B 0.000,C 90.000,E1 20.791} C_DIS
LIN {X -0.137,Y -403.919,Z 810.894,A 0.000,B 0.000,C 90.000,E1 16.968} C_DIS
LIN {X 0.081,Y -409.268,Z 810.873,A 0.000,B 0.000,C 90.000,E1 13.119} C_DIS
LIN {X -0.082,Y -412.690,Z 810.862,A 0.000,B 0.000,C 90.000,E1 11.074} C_DIS
LIN {X -0.166,Y -416.250,Z 810.850,A 0.000,B 0.000,C 90.000,E1 9.029} C_DIS
LIN {X 0.119,Y -420.565,Z 810.837,A 0.000,B 0.000,C 90.000,E1 6.606} C_DIS
LIN {X -0.073,Y -423.047,Z 810.829,A 0.000,B 0.000,C 90.000,E1 5.277} C_DIS
LIN {X -0.097,Y -427.480,Z 810.816,A 0.000,B 0.000,C 90.000,E1 2.922} C_DIS
LIN {X 0.165,Y -433.914,Z 810.799,A 0.000,B 0.000,C 90.000,E1 359.771} C_DIS
LIN {X -0.020,Y -439.016,Z 810.786,A 0.000,B 0.000,C 90.000,E1 357.478} C_DIS
LIN {X -0.173,Y -443.746,Z 810.775,A 0.000,B 0.000,C 90.000,E1 355.527} C_DIS
LIN {X -0.185,Y -448.588,Z 810.764,A 0.000,B 0.000,C 90.000,E1 353.571} C_DIS
LIN {X 0.023,Y -453.482,Z 810.753,A 0.000,B 0.000,C 90.000,E1 351.602} C_DIS
LIN {X -0.094,Y -456.908,Z 810.746,A 0.000,B 0.000,C 90.000,E1 350.330} C_DIS
LIN {X -0.170,Y -458.572,Z 810.744,A 0.000,B 0.000,C 90.000,E1 349.859} C_DIS
LIN {X 0.135,Y -460.856,Z 810.741,A 0.000,B 0.000,C 90.000,E1 349.342} C_DIS
LIN {X -0.133,Y -463.222,Z 810.739,A 0.000,B 0.000,C 90.000,E1 348.993} C_DIS
LIN {X 0.206,Y -465.957,Z 810.737,A 0.000,B 0.000,C 90.000,E1 348.634} C_DIS
LIN {X -0.053,Y -470.470,Z 810.735,A 0.000,B 0.000,C 90.000,E1 348.229} C_DIS
LIN {X -0.108,Y -478.593,Z 810.731,A 0.000,B 0.000,C 90.000,E1 347.589} C_DIS
LIN {X -0.017,Y -493.176,Z 810.726,A 0.000,B 0.000,C 90.000,E1 346.589} C_DIS
LIN {X 0.028,Y -507.355,Z 810.720,A 0.000,B 0.000,C 90.000,E1 345.644} C_DIS
LIN {X -0.099,Y -519.918,Z 810.716,A 0.000,B 0.000,C 90.000,E1 344.810} C_DIS
LIN {X 0.162,Y -532.225,Z 810.711,A 0.000,B 0.000,C 90.000,E1 343.921} C_DIS
LIN {X 0.141,Y -539.740,Z 810.708,A 0.000,B 0.000,C 90.000,E1 343.378} C_DIS
LIN {X -0.084,Y -547.182,Z 810.705,A 0.000,B 0.000,C 90.000,E1 342.834} C_DIS
LIN {X -0.086,Y -555.784,Z 810.701,A 0.000,B 0.000,C 90.000,E1 342.127} C_DIS
LIN {X -0.121,Y -561.203,Z 810.698,A 0.000,B 0.000,C 90.000,E1 341.638} C_DIS
LIN {X 0.243,Y -566.609,Z 810.695,A 0.000,B 0.000,C 90.000,E1 341.094} C_DIS
LIN {X 0.089,Y -574.218,Z 810.691,A 0.000,B 0.000,C 90.000,E1 340.315} C_DIS
LIN {X -0.065,Y -581.059,Z 810.686,A 0.000,B 0.000,C 90.000,E1 339.518} C_DIS
LIN {X 0.184,Y -585.154,Z 810.683,A 0.000,B 0.000,C 90.000,E1 338.954} C_DIS
LIN {X 0.132,Y -590.824,Z 810.679,A 0.000,B 0.000,C 90.000,E1 338.156} C_DIS
LIN {X 0.086,Y -596.968,Z 810.674,A 0.000,B 0.000,C 90.000,E1 337.230} C_DIS
LIN {X 0.147,Y -601.869,Z 810.669,A 0.000,B 0.000,C 90.000,E1 336.433} C_DIS
LIN {X -0.081,Y -607.360,Z 810.664,A 0.000,B 0.000,C 90.000,E1 335.537} C_DIS
LIN {X 0.300,Y -613.457,Z 810.658,A 0.000,B 0.000,C 90.000,E1 334.460} C_DIS
LIN {X -0.055,Y -618.520,Z 810.653,A 0.000,B 0.000,C 90.000,E1 333.589} C_DIS
LIN {X 0.202,Y -623.362,Z 810.648,A 0.000,B 0.000,C 90.000,E1 332.666} C_DIS
LIN {X 0.227,Y -627.286,Z 810.644,A 0.000,B 0.000,C 90.000,E1 331.897} C_DIS
LIN {X -0.213,Y -633.360,Z 810.637,A 0.000,B 0.000,C 90.000,E1 330.667} C_DIS
LIN {X -0.279,Y -638.531,Z 810.631,A 0.000,B 0.000,C 90.000,E1 329.537} C_DIS
LIN {X 0.195,Y -641.858,Z 810.626,A 0.000,B 0.000,C 90.000,E1 328.742} C_DIS
LIN {X 0.157,Y -644.963,Z 810.622,A 0.000,B 0.000,C 90.000,E1 327.995} C_DIS
LIN {X 0.152,Y -647.893,Z 810.618,A 0.000,B 0.000,C 90.000,E1 327.248} C_DIS
LIN {X 0.142,Y -652.462,Z 810.611,A 0.000,B 0.000,C 90.000,E1 326.008} C_DIS
LIN {X 0.123,Y -655.785,Z 810.606,A 0.000,B 0.000,C 90.000,E1 325.022} C_DIS
LIN {X -0.236,Y -658.961,Z 810.600,A 0.000,B 0.000,C 90.000,E1 324.069} C_DIS
LIN {X -0.225,Y -662.551,Z 810.594,A 0.000,B 0.000,C 90.000,E1 322.844} C_DIS
LIN {X -0.154,Y -665.735,Z 810.587,A 0.000,B 0.000,C 90.000,E1 321.618} C_DIS
LIN {X 0.385,Y -668.657,Z 810.580,A 0.000,B 0.000,C 90.000,E1 320.356} C_DIS
LIN {X 0.460,Y -670.873,Z 810.575,A 0.000,B 0.000,C 90.000,E1 319.380} C_DIS
LIN {X -0.374,Y -673.402,Z 810.568,A 0.000,B 0.000,C 90.000,E1 318.243} C_DIS
LIN {X 0.183,Y -674.823,Z 810.564,A 0.000,B 0.000,C 90.000,E1 317.472} C_DIS
LIN {X -0.110,Y -677.319,Z 810.556,A 0.000,B 0.000,C 90.000,E1 316.053} C_DIS
LIN {X 0.036,Y -678.774,Z 810.551,A 0.000,B 0.000,C 90.000,E1 315.081} C_DIS
LIN {X 0.289,Y -680.731,Z 810.543,A 0.000,B 0.000,C 90.000,E1 313.623} C_DIS
LIN {X -0.309,Y -682.761,Z 810.533,A 0.000,B 0.000,C 90.000,E1 312.000} C_DIS
LIN {X 0.000,Y -684.187,Z 810.527,A 0.000,B 0.000,C 90.000,E1 310.782} C_DIS
LIN {X -0.060,Y -685.649,Z 810.519,A 0.000,B 0.000,C 90.000,E1 309.358} C_DIS
LIN {X 0.233,Y -686.582,Z 810.513,A 0.000,B 0.000,C 90.000,E1 308.382} C_DIS
LIN {X -0.049,Y -688.081,Z 810.504,A 0.000,B 0.000,C 90.000,E1 306.744} C_DIS
LIN {X 0.439,Y -689.065,Z 810.498,A 0.000,B 0.000,C 90.000,E1 305.518} C_DIS
LIN {X -0.424,Y -689.985,Z 810.491,A 0.000,B 0.000,C 90.000,E1 304.405} C_DIS
LIN {X 0.119,Y -691.160,Z 810.482,A 0.000,B 0.000,C 90.000,E1 302.704} C_DIS
LIN {X 0.333,Y -692.619,Z 810.471,A 0.000,B 0.000,C 90.000,E1 300.797} C_DIS
LIN {X -0.266,Y -693.424,Z 810.465,A 0.000,B 0.000,C 90.000,E1 299.667} C_DIS
LIN {X -0.117,Y -694.668,Z 810.454,A 0.000,B 0.000,C 90.000,E1 297.769} C_DIS
LIN {X -0.014,Y -696.169,Z 810.443,A 0.000,B 0.000,C 90.000,E1 295.643} C_DIS
LIN {X -0.208,Y -696.861,Z 810.437,A 0.000,B 0.000,C 90.000,E1 294.719} C_DIS
LIN {X 0.308,Y -697.082,Z 810.435,A 0.000,B 0.000,C 90.000,E1 294.207} C_DIS
LIN {X -0.096,Y -696.844,Z 810.432,A 0.000,B 0.000,C 90.000,E1 293.770} C_DIS
LIN {X 0.161,Y -696.473,Z 810.431,A 0.000,B 0.000,C 90.000,E1 293.515} C_DIS
LIN {X -0.245,Y -694.844,Z 810.428,A 0.000,B 0.000,C 90.000,E1 293.078} C_DIS
LIN {X -0.120,Y -694.349,Z 810.427,A 0.000,B 0.000,C 90.000,E1 292.950} C_DIS
LIN {X 0.004,Y -693.605,Z 810.427,A 0.000,B 0.000,C 90.000,E1 292.823} C_DIS
LIN {X 0.125,Y -692.495,Z 810.426,A 0.000,B 0.000,C 90.000,E1 292.695} C_DIS
LIN {X -0.152,Y -688.401,Z 810.424,A 0.000,B 0.000,C 90.000,E1 292.386} C_DIS
LIN {X -0.165,Y -686.945,Z 810.424,A 0.000,B 0.000,C 90.000,E1 292.280} C_DIS
LIN {X 0.083,Y -685.022,Z 810.423,A 0.000,B 0.000,C 90.000,E1 292.153} C_DIS
LIN {X 0.200,Y -680.547,Z 810.422,A 0.000,B 0.000,C 90.000,E1 291.972} C_DIS
LIN {X 0.189,Y -675.017,Z 810.421,A 0.000,B 0.000,C 90.000,E1 291.791} C_DIS
LIN {X -0.242,Y -673.059,Z 810.421,A 0.000,B 0.000,C 90.000,E1 291.770} C_DIS
LIN {X -0.196,Y -667.589,Z 810.420,A 0.000,B 0.000,C 90.000,E1 291.663} C_DIS
LIN {X 0.182,Y -645.923,Z 810.418,A 0.000,B 0.000,C 90.000,E1 291.280} C_DIS
LIN {X -0.083,Y -628.436,Z 810.417,A 0.000,B 0.000,C 90.000,E1 290.972} C_DIS
LIN {X -0.057,Y -615.053,Z 810.415,A 0.000,B 0.000,C 90.000,E1 290.663} C_DIS
LIN {X 0.006,Y -607.229,Z 810.414,A 0.000,B 0.000,C 90.000,E1 290.429} C_DIS
LIN {X 0.127,Y -604.066,Z 810.413,A 0.000,B 0.000,C 90.000,E1 290.301} C_DIS
LIN {X -0.015,Y -600.896,Z 810.412,A 0.000,B 0.000,C 90.000,E1 290.174} C_DIS
LIN {X -0.351,Y -597.292,Z 810.411,A 0.000,B 0.000,C 90.000,E1 290.066} C_DIS
LIN {X -0.151,Y -593.465,Z 810.410,A 0.000,B 0.000,C 90.000,E1 289.812} C_DIS
LIN {X -0.102,Y -592.437,Z 810.410,A 0.000,B 0.000,C 90.000,E1 289.758} C_DIS
LIN {X 0.212,Y -591.216,Z 810.409,A 0.000,B 0.000,C 90.000,E1 289.631} C_DIS
LIN {X -0.329,Y -590.249,Z 810.409,A 0.000,B 0.000,C 90.000,E1 289.577} C_DIS
LIN {X 0.177,Y -590.236,Z 810.409,A 0.000,B 0.000,C 90.000,E1 289.523} C_DIS
LIN {X 0.161,Y -590.390,Z 810.407,A 0.000,B 0.000,C 90.000,E1 289.214} C_DIS
LIN {X 0.097,Y -590.787,Z 810.406,A 0.000,B 0.000,C 90.000,E1 289.087} C_DIS
LIN {X -0.285,Y -592.618,Z 810.404,A 0.000,B 0.000,C 90.000,E1 288.725} C_DIS
LIN {X 0.198,Y -599.884,Z 810.397,A 0.000,B 0.000,C 90.000,E1 287.511} C_DIS
LIN {X 0.199,Y -602.728,Z 810.395,A 0.000,B 0.000,C 90.000,E1 286.985} C_DIS
LIN {X 0.348,Y -605.774,Z 810.391,A 0.000,B 0.000,C 90.000,E1 286.315} C_DIS
LIN {X -0.189,Y -607.835,Z 810.388,A 0.000,B 0.000,C 90.000,E1 285.843} C_DIS
LIN {X 0.132,Y -608.726,Z 810.387,A 0.000,B 0.000,C 90.000,E1 285.552} C_DIS
LIN {X -0.223,Y -610.082,Z 810.384,A 0.000,B 0.000,C 90.000,E1 285.064} C_DIS
LIN {X -0.141,Y -611.213,Z 810.381,A 0.000,B 0.000,C 90.000,E1 284.537} C_DIS
LIN {X 0.200,Y -611.661,Z 810.379,A 0.000,B 0.000,C 90.000,E1 284.245} C_DIS
LIN {X 0.055,Y -612.269,Z 810.375,A 0.000,B 0.000,C 90.000,E1 283.480} C_DIS
LIN {X -0.190,Y -612.412,Z 810.374,A 0.000,B 0.000,C 90.000,E1 283.244} C_DIS
LIN {X 0.299,Y -612.386,Z 810.372,A 0.000,B 0.000,C 90.000,E1 282.939} C_DIS
LIN {X -0.327,Y -611.891,Z 810.369,A 0.000,B 0.000,C 90.000,E1 282.479} C_DIS
LIN {X -0.221,Y -611.070,Z 810.366,A 0.000,B 0.000,C 90.000,E1 281.951} C_DIS
LIN {X -0.122,Y -609.764,Z 810.363,A 0.000,B 0.000,C 90.000,E1 281.422} C_DIS
LIN {X 0.223,Y -608.919,Z 810.362,A 0.000,B 0.000,C 90.000,E1 281.130} C_DIS
LIN {X 0.041,Y -605.828,Z 810.358,A 0.000,B 0.000,C 90.000,E1 280.366} C_DIS
LIN {X -0.332,Y -604.701,Z 810.356,A 0.000,B 0.000,C 90.000,E1 280.141} C_DIS
LIN {X -0.281,Y -601.915,Z 810.353,A 0.000,B 0.000,C 90.000,E1 279.613} C_DIS
LIN {X 0.333,Y -598.462,Z 810.350,A 0.000,B 0.000,C 90.000,E1 279.029} C_DIS
LIN {X 0.259,Y -594.006,Z 810.347,A 0.000,B 0.000,C 90.000,E1 278.511} C_DIS
LIN {X 0.061,Y -592.754,Z 810.347,A 0.000,B 0.000,C 90.000,E1 278.398} C_DIS
LIN {X -0.128,Y -589.759,Z 810.345,A 0.000,B 0.000,C 90.000,E1 278.163} C_DIS
LIN {X -0.165,Y -586.722,Z 810.344,A 0.000,B 0.000,C 90.000,E1 277.936} C_DIS
LIN {X 0.100,Y -583.321,Z 810.343,A 0.000,B 0.000,C 90.000,E1 277.701} C_DIS
LIN {X -0.245,Y -576.003,Z 810.341,A 0.000,B 0.000,C 90.000,E1 277.409} C_DIS
LIN {X -0.200,Y -569.895,Z 810.340,A 0.000,B 0.000,C 90.000,E1 277.239} C_DIS
LIN {X 0.021,Y -562.820,Z 810.340,A 0.000,B 0.000,C 90.000,E1 277.125} C_DIS
LIN {X -0.245,Y -557.897,Z 810.339,A 0.000,B 0.000,C 90.000,E1 277.125} C_DIS
LIN {X 0.042,Y -555.722,Z 810.339,A 0.000,B 0.000,C 90.000,E1 277.068} C_DIS
LIN {X -0.011,Y -553.244,Z 810.339,A 0.000,B 0.000,C 90.000,E1 277.004} C_DIS
LIN {X -0.042,Y -553.222,Z 810.339,A 0.000,B 0.000,C 90.000,E1 277.004} C_DIS
LIN {X -0.218,Y -550.688,Z 810.337,A 0.000,B 0.000,C 90.000,E1 276.606} C_DIS
LIN {X -0.260,Y -550.668,Z 810.337,A 0.000,B 0.000,C 90.000,E1 276.606} C_DIS
LIN {X 0.116,Y -549.953,Z 810.332,A 0.000,B 0.000,C 90.000,E1 275.796} C_DIS
LIN {X -0.111,Y -549.317,Z 810.325,A 0.000,B 0.000,C 90.000,E1 274.416} C_DIS
LIN {X 0.069,Y -548.822,Z 810.320,A 0.000,B 0.000,C 90.000,E1 273.555} C_DIS
LIN {X -0.211,Y -547.860,Z 810.312,A 0.000,B 0.000,C 90.000,E1 272.178} C_DIS
LIN {X 0.083,Y -546.697,Z 810.303,A 0.000,B 0.000,C 90.000,E1 270.458} C_DIS
LIN {X -0.170,Y -545.318,Z 810.292,A 0.000,B 0.000,C 90.000,E1 268.511} C_DIS
LIN {X 0.150,Y -543.802,Z 810.279,A 0.000,B 0.000,C 90.000,E1 266.216} C_DIS
LIN {X -0.186,Y -542.956,Z 810.271,A 0.000,B 0.000,C 90.000,E1 264.837} C_DIS
LIN {X -0.012,Y -542.165,Z 810.265,A 0.000,B 0.000,C 90.000,E1 263.685} C_DIS
LIN {X 0.216,Y -540.979,Z 810.257,A 0.000,B 0.000,C 90.000,E1 262.243} C_DIS
LIN {X -0.108,Y -540.044,Z 810.251,A 0.000,B 0.000,C 90.000,E1 261.141} C_DIS
LIN {X 0.088,Y -539.007,Z 810.244,A 0.000,B 0.000,C 90.000,E1 259.982} C_DIS
LIN {X 0.029,Y -537.048,Z 810.233,A 0.000,B 0.000,C 90.000,E1 257.993} C_DIS
LIN {X -0.014,Y -535.279,Z 810.224,A 0.000,B 0.000,C 90.000,E1 256.284} C_DIS
LIN {X -0.098,Y -533.342,Z 810.214,A 0.000,B 0.000,C 90.000,E1 254.574} C_DIS
LIN {X -0.127,Y -531.678,Z 810.206,A 0.000,B 0.000,C 90.000,E1 253.142} C_DIS
LIN {X -0.026,Y -529.985,Z 810.198,A 0.000,B 0.000,C 90.000,E1 251.692} C_DIS
LIN {X 0.044,Y -528.155,Z 810.190,A 0.000,B 0.000,C 90.000,E1 250.242} C_DIS
LIN {X 0.081,Y -526.600,Z 810.184,A 0.000,B 0.000,C 90.000,E1 249.082} C_DIS
LIN {X 0.102,Y -523.692,Z 810.173,A 0.000,B 0.000,C 90.000,E1 247.050} C_DIS
LIN {X 0.086,Y -521.067,Z 810.163,A 0.000,B 0.000,C 90.000,E1 245.305} C_DIS
LIN {X -0.194,Y -519.678,Z 810.158,A 0.000,B 0.000,C 90.000,E1 244.460} C_DIS
LIN {X 0.150,Y -516.646,Z 810.148,A 0.000,B 0.000,C 90.000,E1 242.666} C_DIS
LIN {X 0.293,Y -515.124,Z 810.143,A 0.000,B 0.000,C 90.000,E1 241.769} C_DIS
LIN {X -0.036,Y -512.394,Z 810.135,A 0.000,B 0.000,C 90.000,E1 240.333} C_DIS
LIN {X -0.160,Y -509.617,Z 810.127,A 0.000,B 0.000,C 90.000,E1 238.869} C_DIS
LIN {X -0.067,Y -506.573,Z 810.119,A 0.000,B 0.000,C 90.000,E1 237.375} C_DIS
LIN {X -0.035,Y -503.429,Z 810.110,A 0.000,B 0.000,C 90.000,E1 235.881} C_DIS
LIN {X -0.196,Y -500.148,Z 810.102,A 0.000,B 0.000,C 90.000,E1 234.402} C_DIS
LIN {X 0.278,Y -496.429,Z 810.094,A 0.000,B 0.000,C 90.000,E1 232.844} C_DIS
LIN {X 0.035,Y -493.498,Z 810.087,A 0.000,B 0.000,C 90.000,E1 231.662} C_DIS
LIN {X -0.021,Y -489.728,Z 810.079,A 0.000,B 0.000,C 90.000,E1 230.150} C_DIS
LIN {X 0.069,Y -484.812,Z 810.067,A 0.000,B 0.000,C 90.000,E1 228.000} C_DIS
LIN {X -0.319,Y -480.104,Z 810.055,A 0.000,B 0.000,C 90.000,E1 225.891} C_DIS
LIN {X -0.276,Y -476.030,Z 810.044,A 0.000,B 0.000,C 90.000,E1 224.028} C_DIS
LIN {X -0.132,Y -470.631,Z 810.031,A 0.000,B 0.000,C 90.000,E1 221.515} C_DIS
LIN {X -0.014,Y -467.322,Z 810.022,A 0.000,B 0.000,C 90.000,E1 219.930} C_DIS
LIN {X 0.108,Y -464.070,Z 810.013,A 0.000,B 0.000,C 90.000,E1 218.338} C_DIS
LIN {X -0.064,Y -459.424,Z 810.001,A 0.000,B 0.000,C 90.000,E1 216.137} C_DIS
LIN {X 0.001,Y -456.132,Z 809.992,A 0.000,B 0.000,C 90.000,E1 214.532} C_DIS
LIN {X -0.059,Y -451.564,Z 809.979,A 0.000,B 0.000,C 90.000,E1 212.291} C_DIS
LIN {X 0.143,Y -446.907,Z 809.967,A 0.000,B 0.000,C 90.000,E1 210.001} C_DIS
LIN {X 0.194,Y -444.331,Z 809.960,A 0.000,B 0.000,C 90.000,E1 208.693} C_DIS
LIN {X 0.091,Y -440.530,Z 809.949,A 0.000,B 0.000,C 90.000,E1 206.744} C_DIS
LIN {X 0.073,Y -437.412,Z 809.940,A 0.000,B 0.000,C 90.000,E1 205.103} C_DIS
LIN {X 0.217,Y -432.837,Z 809.927,A 0.000,B 0.000,C 90.000,E1 202.770} C_DIS
LIN {X 0.079,Y -428.935,Z 809.916,A 0.000,B 0.000,C 90.000,E1 200.791} C_DIS
LIN {X 0.095,Y -425.114,Z 809.904,A 0.000,B 0.000,C 90.000,E1 198.779} C_DIS
LIN {X 0.102,Y -421.874,Z 809.895,A 0.000,B 0.000,C 90.000,E1 197.094} C_DIS
LIN {X 0.135,Y -417.305,Z 809.882,A 0.000,B 0.000,C 90.000,E1 194.717} C_DIS
LIN {X -0.062,Y -412.765,Z 809.869,A 0.000,B 0.000,C 90.000,E1 192.355} C_DIS
LIN {X 0.190,Y -409.605,Z 809.859,A 0.000,B 0.000,C 90.000,E1 190.602} C_DIS
LIN {X -0.084,Y -405.761,Z 809.848,A 0.000,B 0.000,C 90.000,E1 188.568} C_DIS
LIN {X -0.162,Y -401.280,Z 809.834,A 0.000,B 0.000,C 90.000,E1 186.144} C_DIS
LIN {X 0.080,Y -398.249,Z 809.824,A 0.000,B 0.000,C 90.000,E1 184.359} C_DIS
LIN {X -0.028,Y -393.558,Z 809.807,A 0.000,B 0.000,C 90.000,E1 181.203} C_DIS
LIN {X -0.082,Y -390.863,Z 809.795,A 0.000,B 0.000,C 90.000,E1 179.083} C_DIS
LIN {X 0.120,Y -388.080,Z 809.781,A 0.000,B 0.000,C 90.000,E1 176.560} C_DIS
LIN {X 0.183,Y -384.917,Z 809.765,A 0.000,B 0.000,C 90.000,E1 173.685} C_DIS
LIN {X 0.054,Y -382.675,Z 809.753,A 0.000,B 0.000,C 90.000,E1 171.546} C_DIS
LIN {X 0.103,Y -381.378,Z 809.745,A 0.000,B 0.000,C 90.000,E1 170.095} C_DIS
LIN {X -0.101,Y -378.862,Z 809.729,A 0.000,B 0.000,C 90.000,E1 167.229} C_DIS
LIN {X 0.146,Y -376.729,Z 809.713,A 0.000,B 0.000,C 90.000,E1 164.283} C_DIS
LIN {X -0.101,Y -375.318,Z 809.697,A 0.000,B 0.000,C 90.000,E1 161.402} C_DIS
LIN {X 0.134,Y -374.935,Z 809.670,A 0.000,B 0.000,C 90.000,E1 156.613} C_DIS
LIN {X -0.039,Y -376.349,Z 809.654,A 0.000,B 0.000,C 90.000,E1 153.717} C_DIS
LIN {X 0.010,Y -377.441,Z 809.648,A 0.000,B 0.000,C 90.000,E1 152.615} C_DIS
LIN {X 0.018,Y -379.814,Z 809.638,A 0.000,B 0.000,C 90.000,E1 150.795} C_DIS
LIN {X -0.030,Y -382.008,Z 809.632,A 0.000,B 0.000,C 90.000,E1 149.715} C_DIS
LIN {X -0.064,Y -383.841,Z 809.628,A 0.000,B 0.000,C 90.000,E1 148.997} C_DIS
LIN {X 0.091,Y -386.772,Z 809.623,A 0.000,B 0.000,C 90.000,E1 148.074} C_DIS
LIN {X -0.023,Y -389.945,Z 809.618,A 0.000,B 0.000,C 90.000,E1 147.296} C_DIS
LIN {X 0.005,Y -391.250,Z 809.617,A 0.000,B 0.000,C 90.000,E1 147.041} C_DIS
LIN {X 0.051,Y -393.657,Z 809.614,A 0.000,B 0.000,C 90.000,E1 146.501} C_DIS
LIN {X -0.012,Y -397.361,Z 809.610,A 0.000,B 0.000,C 90.000,E1 145.801} C_DIS
LIN {X 0.184,Y -402.611,Z 809.606,A 0.000,B 0.000,C 90.000,E1 144.975} C_DIS
LIN {X -0.034,Y -406.523,Z 809.603,A 0.000,B 0.000,C 90.000,E1 144.482} C_DIS
LIN {X 0.247,Y -413.461,Z 809.598,A 0.000,B 0.000,C 90.000,E1 143.623} C_DIS
LIN {X -0.145,Y -419.288,Z 809.595,A 0.000,B 0.000,C 90.000,E1 143.050} C_DIS
LIN {X 0.107,Y -424.832,Z 809.592,A 0.000,B 0.000,C 90.000,E1 142.477} C_DIS
LIN {X 0.092,Y -429.095,Z 809.589,A 0.000,B 0.000,C 90.000,E1 142.029} C_DIS
LIN {X 0.045,Y -435.859,Z 809.585,A 0.000,B 0.000,C 90.000,E1 141.251} C_DIS
LIN {X 0.247,Y -446.397,Z 809.578,A 0.000,B 0.000,C 90.000,E1 139.989} C_DIS
LIN {X 0.010,Y -450.253,Z 809.575,A 0.000,B 0.000,C 90.000,E1 139.542} C_DIS
LIN {X -0.059,Y -456.462,Z 809.571,A 0.000,B 0.000,C 90.000,E1 138.771} C_DIS
LIN {X 0.046,Y -462.157,Z 809.567,A 0.000,B 0.000,C 90.000,E1 137.957} C_DIS
LIN {X 0.209,Y -468.621,Z 809.561,A 0.000,B 0.000,C 90.000,E1 136.986} C_DIS
LIN {X 0.083,Y -473.360,Z 809.557,A 0.000,B 0.000,C 90.000,E1 136.215} C_DIS
LIN {X -0.292,Y -484.944,Z 809.546,A 0.000,B 0.000,C 90.000,E1 134.271} C_DIS
LIN {X -0.081,Y -487.601,Z 809.543,A 0.000,B 0.000,C 90.000,E1 133.785} C_DIS
LIN {X 0.224,Y -494.335,Z 809.536,A 0.000,B 0.000,C 90.000,E1 132.528} C_DIS
LIN {X 0.251,Y -497.616,Z 809.533,A 0.000,B 0.000,C 90.000,E1 131.919} C_DIS
LIN {X -0.304,Y -501.261,Z 809.529,A 0.000,B 0.000,C 90.000,E1 131.229} C_DIS
LIN {X -0.002,Y -503.599,Z 809.526,A 0.000,B 0.000,C 90.000,E1 130.744} C_DIS
LIN {X -0.231,Y -508.419,Z 809.521,A 0.000,B 0.000,C 90.000,E1 129.725} C_DIS
LIN {X -0.101,Y -511.416,Z 809.517,A 0.000,B 0.000,C 90.000,E1 129.116} C_DIS
LIN {X -0.189,Y -512.801,Z 809.516,A 0.000,B 0.000,C 90.000,E1 128.830} C_DIS
LIN {X -0.151,Y -514.573,Z 809.513,A 0.000,B 0.000,C 90.000,E1 128.382} C_DIS
LIN {X -0.079,Y -517.176,Z 809.510,A 0.000,B 0.000,C 90.000,E1 127.855} C_DIS
LIN {X 0.265,Y -518.513,Z 809.509,A 0.000,B 0.000,C 90.000,E1 127.523} C_DIS
LIN {X 0.148,Y -520.913,Z 809.505,A 0.000,B 0.000,C 90.000,E1 126.950} C_DIS
LIN {X -0.142,Y -523.233,Z 809.503,A 0.000,B 0.000,C 90.000,E1 126.457} C_DIS
LIN {X -0.184,Y -524.511,Z 809.501,A 0.000,B 0.000,C 90.000,E1 126.171} C_DIS
LIN {X -0.294,Y -527.802,Z 809.496,A 0.000,B 0.000,C 90.000,E1 125.311} C_DIS
LIN {X 0.108,Y -528.845,Z 809.494,A 0.000,B 0.000,C 90.000,E1 124.978} C_DIS
LIN {X 0.083,Y -529.499,Z 809.493,A 0.000,B 0.000,C 90.000,E1 124.692} C_DIS
LIN {X 0.039,Y -531.419,Z 809.490,A 0.000,B 0.000,C 90.000,E1 124.119} C_DIS
LIN {X 0.020,Y -532.212,Z 809.488,A 0.000,B 0.000,C 90.000,E1 123.833} C_DIS
LIN {X -0.091,Y -537.719,Z 809.480,A 0.000,B 0.000,C 90.000,E1 122.418} C_DIS
LIN {X 0.087,Y -540.885,Z 809.475,A 0.000,B 0.000,C 90.000,E1 121.544} C_DIS
LIN {X -0.167,Y -543.761,Z 809.471,A 0.000,B 0.000,C 90.000,E1 120.718} C_DIS
LIN {X -0.202,Y -546.404,Z 809.466,A 0.000,B 0.000,C 90.000,E1 119.873} C_DIS
LIN {X -0.179,Y -549.731,Z 809.460,A 0.000,B 0.000,C 90.000,E1 118.743} C_DIS
LIN {X -0.145,Y -552.005,Z 809.455,A 0.000,B 0.000,C 90.000,E1 117.897} C_DIS
LIN {X -0.089,Y -553.994,Z 809.450,A 0.000,B 0.000,C 90.000,E1 117.052} C_DIS
LIN {X -0.261,Y -555.676,Z 809.446,A 0.000,B 0.000,C 90.000,E1 116.232} C_DIS
LIN {X -0.195,Y -556.668,Z 809.443,A 0.000,B 0.000,C 90.000,E1 115.668} C_DIS
LIN {X 0.197,Y -558.285,Z 809.436,A 0.000,B 0.000,C 90.000,E1 114.515} C_DIS
LIN {X -0.052,Y -560.067,Z 809.429,A 0.000,B 0.000,C 90.000,E1 113.153} C_DIS
LIN {X -0.157,Y -560.990,Z 809.424,A 0.000,B 0.000,C 90.000,E1 112.333} C_DIS
LIN {X -0.153,Y -562.053,Z 809.418,A 0.000,B 0.000,C 90.000,E1 111.227} C_DIS
LIN {X -0.135,Y -562.734,Z 809.412,A 0.000,B 0.000,C 90.000,E1 110.120} C_DIS
LIN {X -0.115,Y -563.231,Z 809.406,A 0.000,B 0.000,C 90.000,E1 109.014} C_DIS
LIN {X 0.257,Y -563.550,Z 809.399,A 0.000,B 0.000,C 90.000,E1 107.873} C_DIS
LIN {X 0.013,Y -564.208,Z 809.389,A 0.000,B 0.000,C 90.000,E1 105.969} C_DIS
LIN {X -0.209,Y -565.132,Z 809.378,A 0.000,B 0.000,C 90.000,E1 104.064} C_DIS
LIN {X 0.163,Y -566.539,Z 809.366,A 0.000,B 0.000,C 90.000,E1 101.827} C_DIS
LIN {X 0.167,Y -567.916,Z 809.355,A 0.000,B 0.000,C 90.000,E1 99.905} C_DIS
LIN {X 0.020,Y -569.130,Z 809.346,A 0.000,B 0.000,C 90.000,E1 98.276} C_DIS
LIN {X 0.192,Y -570.042,Z 809.338,A 0.000,B 0.000,C 90.000,E1 96.891} C_DIS
LIN {X 0.049,Y -571.116,Z 809.328,A 0.000,B 0.000,C 90.000,E1 94.992} C_DIS
LIN {X 0.202,Y -571.760,Z 809.320,A 0.000,B 0.000,C 90.000,E1 93.612} C_DIS
LIN {X 0.195,Y -572.220,Z 809.314,A 0.000,B 0.000,C 90.000,E1 92.522} C_DIS
LIN {X 0.035,Y -572.938,Z 809.304,A 0.000,B 0.000,C 90.000,E1 90.630} C_DIS
LIN {X -0.262,Y -573.454,Z 809.294,A 0.000,B 0.000,C 90.000,E1 89.026} C_DIS
LIN {X 0.036,Y -573.865,Z 809.285,A 0.000,B 0.000,C 90.000,E1 87.364} C_DIS
LIN {X -0.199,Y -574.217,Z 809.276,A 0.000,B 0.000,C 90.000,E1 85.755} C_DIS
LIN {X 0.010,Y -574.504,Z 809.269,A 0.000,B 0.000,C 90.000,E1 84.375} C_DIS
LIN {X 0.088,Y -574.749,Z 809.263,A 0.000,B 0.000,C 90.000,E1 83.280} C_DIS
LIN {X 0.114,Y -575.137,Z 809.252,A 0.000,B 0.000,C 90.000,E1 81.376} C_DIS
LIN {X 0.116,Y -575.489,Z 809.243,A 0.000,B 0.000,C 90.000,E1 79.746} C_DIS
LIN {X -0.085,Y -575.798,Z 809.236,A 0.000,B 0.000,C 90.000,E1 78.409} C_DIS
LIN {X 0.167,Y -575.933,Z 809.227,A 0.000,B 0.000,C 90.000,E1 76.756} C_DIS
LIN {X -0.122,Y -575.923,Z 809.221,A 0.000,B 0.000,C 90.000,E1 75.700} C_DIS
LIN {X 0.286,Y -575.882,Z 809.215,A 0.000,B 0.000,C 90.000,E1 74.574} C_DIS
LIN {X 0.141,Y -575.746,Z 809.205,A 0.000,B 0.000,C 90.000,E1 72.960} C_DIS
LIN {X 0.169,Y -575.453,Z 809.196,A 0.000,B 0.000,C 90.000,E1 71.329} C_DIS
LIN {X -0.183,Y -575.081,Z 809.189,A 0.000,B 0.000,C 90.000,E1 70.007} C_DIS
LIN {X 0.016,Y -574.759,Z 809.183,A 0.000,B 0.000,C 90.000,E1 68.901} C_DIS
LIN {X 0.049,Y -574.274,Z 809.175,A 0.000,B 0.000,C 90.000,E1 67.539} C_DIS
LIN {X -0.090,Y -573.515,Z 809.166,A 0.000,B 0.000,C 90.000,E1 65.921} C_DIS
LIN {X 0.145,Y -572.810,Z 809.159,A 0.000,B 0.000,C 90.000,E1 64.537} C_DIS
LIN {X 0.103,Y -571.947,Z 809.151,A 0.000,B 0.000,C 90.000,E1 63.179} C_DIS
LIN {X 0.120,Y -571.259,Z 809.147,A 0.000,B 0.000,C 90.000,E1 62.359} C_DIS
LIN {X 0.047,Y -569.895,Z 809.139,A 0.000,B 0.000,C 90.000,E1 61.001} C_DIS
LIN {X -0.090,Y -568.635,Z 809.133,A 0.000,B 0.000,C 90.000,E1 59.921} C_DIS
LIN {X -0.040,Y -567.133,Z 809.127,A 0.000,B 0.000,C 90.000,E1 58.820} C_DIS
LIN {X 0.091,Y -565.392,Z 809.121,A 0.000,B 0.000,C 90.000,E1 57.709} C_DIS
LIN {X -0.201,Y -563.947,Z 809.116,A 0.000,B 0.000,C 90.000,E1 56.914} C_DIS
LIN {X -0.104,Y -561.744,Z 809.110,A 0.000,B 0.000,C 90.000,E1 55.801} C_DIS
LIN {X -0.131,Y -559.906,Z 809.105,A 0.000,B 0.000,C 90.000,E1 54.975} C_DIS
LIN {X 0.145,Y -557.835,Z 809.101,A 0.000,B 0.000,C 90.000,E1 54.116} C_DIS
LIN {X 0.069,Y -555.544,Z 809.096,A 0.000,B 0.000,C 90.000,E1 53.290} C_DIS
LIN {X -0.146,Y -552.927,Z 809.091,A 0.000,B 0.000,C 90.000,E1 52.477} C_DIS
LIN {X -0.009,Y -551.115,Z 809.088,A 0.000,B 0.000,C 90.000,E1 51.904} C_DIS
LIN {X -0.262,Y -547.987,Z 809.084,A 0.000,B 0.000,C 90.000,E1 51.090} C_DIS
LIN {X 0.225,Y -544.580,Z 809.079,A 0.000,B 0.000,C 90.000,E1 50.194} C_DIS
LIN {X -0.284,Y -541.472,Z 809.075,A 0.000,B 0.000,C 90.000,E1 49.542} C_DIS
LIN {X 0.107,Y -538.711,Z 809.072,A 0.000,B 0.000,C 90.000,E1 48.933} C_DIS
LIN {X 0.072,Y -535.765,Z 809.069,A 0.000,B 0.000,C 90.000,E1 48.366} C_DIS
LIN {X 0.231,Y -531.529,Z 809.065,A 0.000,B 0.000,C 90.000,E1 47.634} C_DIS
LIN {X -0.016,Y -528.854,Z 809.062,A 0.000,B 0.000,C 90.000,E1 47.229} C_DIS
LIN {X 0.047,Y -523.731,Z 809.058,A 0.000,B 0.000,C 90.000,E1 46.500} C_DIS
LIN {X 0.291,Y -519.258,Z 809.055,A 0.000,B 0.000,C 90.000,E1 45.891} C_DIS
LIN {X -0.012,Y -515.685,Z 809.053,A 0.000,B 0.000,C 90.000,E1 45.486} C_DIS
LIN {X -0.148,Y -510.484,Z 809.049,A 0.000,B 0.000,C 90.000,E1 44.919} C_DIS
LIN {X -0.028,Y -506.471,Z 809.047,A 0.000,B 0.000,C 90.000,E1 44.474} C_DIS
LIN {X -0.073,Y -499.326,Z 809.043,A 0.000,B 0.000,C 90.000,E1 43.785} C_DIS
LIN {X -0.055,Y -494.992,Z 809.041,A 0.000,B 0.000,C 90.000,E1 43.380} C_DIS
LIN {X 0.055,Y -490.496,Z 809.039,A 0.000,B 0.000,C 90.000,E1 42.975} C_DIS
LIN {X -0.037,Y -484.276,Z 809.036,A 0.000,B 0.000,C 90.000,E1 42.486} C_DIS
LIN {X 0.033,Y -478.058,Z 809.033,A 0.000,B 0.000,C 90.000,E1 42.000} C_DIS
LIN {X 0.001,Y -468.541,Z 809.030,A 0.000,B 0.000,C 90.000,E1 41.310} C_DIS
LIN {X 0.193,Y -455.736,Z 809.024,A 0.000,B 0.000,C 90.000,E1 40.378} C_DIS
LIN {X 0.279,Y -444.519,Z 809.020,A 0.000,B 0.000,C 90.000,E1 39.564} C_DIS
LIN {X 0.149,Y -421.098,Z 809.010,A 0.000,B 0.000,C 90.000,E1 37.810} C_DIS
LIN {X -0.042,Y -410.475,Z 809.005,A 0.000,B 0.000,C 90.000,E1 36.950} C_DIS
LIN {X 0.031,Y -403.813,Z 809.002,A 0.000,B 0.000,C 90.000,E1 36.297} C_DIS
LIN {X -0.133,Y -402.310,Z 809.001,A 0.000,B 0.000,C 90.000,E1 36.171} C_DIS
LIN {X 0.053,Y -400.531,Z 809.000,A 0.000,B 0.000,C 90.000,E1 35.931} C_DIS
LIN {X 0.016,Y -400.499,Z 809.000,A 0.000,B 0.000,C 90.000,E1 35.931} C_DIS
LIN {X -0.021,Y -393.638,Z 808.976,A 0.000,B 0.000,C 90.000,E1 31.750} C_DIS
LIN {X -0.228,Y -394.758,Z 808.961,A 0.000,B 0.000,C 90.000,E1 28.949} C_DIS
LIN {X -0.095,Y -396.331,Z 808.945,A 0.000,B 0.000,C 90.000,E1 26.104} C_DIS
LIN {X -0.129,Y -397.965,Z 808.931,A 0.000,B 0.000,C 90.000,E1 23.643} C_DIS
LIN {X 0.164,Y -400.162,Z 808.916,A 0.000,B 0.000,C 90.000,E1 20.791} C_DIS
LIN {X -0.087,Y -403.742,Z 808.896,A 0.000,B 0.000,C 90.000,E1 17.330} C_DIS
LIN {X 0.127,Y -408.965,Z 808.875,A 0.000,B 0.000,C 90.000,E1 13.480} C_DIS
LIN {X 0.082,Y -412.942,Z 808.862,A 0.000,B 0.000,C 90.000,E1 11.074} C_DIS
LIN {X 0.054,Y -417.048,Z 808.848,A 0.000,B 0.000,C 90.000,E1 8.681} C_DIS
LIN {X -0.120,Y -420.791,Z 808.837,A 0.000,B 0.000,C 90.000,E1 6.663} C_DIS
LIN {X 0.110,Y -423.277,Z 808.829,A 0.000,B 0.000,C 90.000,E1 5.277} C_DIS
LIN {X 0.095,Y -427.679,Z 808.816,A 0.000,B 0.000,C 90.000,E1 2.922} C_DIS
LIN {X 0.165,Y -432.411,Z 808.803,A 0.000,B 0.000,C 90.000,E1 0.573} C_DIS
LIN {X 0.005,Y -436.296,Z 808.793,A 0.000,B 0.000,C 90.000,E1 358.797} C_DIS
LIN {X 0.015,Y -442.358,Z 808.779,A 0.000,B 0.000,C 90.000,E1 356.159} C_DIS
LIN {X -0.029,Y -447.191,Z 808.768,A 0.000,B 0.000,C 90.000,E1 354.204} C_DIS
LIN {X 0.205,Y -450.390,Z 808.761,A 0.000,B 0.000,C 90.000,E1 352.875} C_DIS
LIN {X 0.255,Y -454.462,Z 808.752,A 0.000,B 0.000,C 90.000,E1 351.254} C_DIS
LIN {X -0.069,Y -456.987,Z 808.746,A 0.000,B 0.000,C 90.000,E1 350.330} C_DIS
LIN {X -0.145,Y -458.555,Z 808.744,A 0.000,B 0.000,C 90.000,E1 349.859} C_DIS
LIN {X 0.086,Y -459.994,Z 808.742,A 0.000,B 0.000,C 90.000,E1 349.511} C_DIS
LIN {X -0.129,Y -461.324,Z 808.740,A 0.000,B 0.000,C 90.000,E1 349.218} C_DIS
LIN {X 0.191,Y -464.399,Z 808.737,A 0.000,B 0.000,C 90.000,E1 348.701} C_DIS
LIN {X -0.113,Y -468.627,Z 808.735,A 0.000,B 0.000,C 90.000,E1 348.285} C_DIS
LIN {X 0.185,Y -471.255,Z 808.733,A 0.000,B 0.000,C 90.000,E1 347.993} C_DIS
LIN {X -0.006,Y -478.031,Z 808.730,A 0.000,B 0.000,C 90.000,E1 347.465} C_DIS
LIN {X 0.186,Y -490.434,Z 808.726,A 0.000,B 0.000,C 90.000,E1 346.589} C_DIS
LIN {X 0.282,Y -506.207,Z 808.720,A 0.000,B 0.000,C 90.000,E1 345.519} C_DIS
LIN {X 0.065,Y -518.789,Z 808.715,A 0.000,B 0.000,C 90.000,E1 344.700} C_DIS
LIN {X -0.174,Y -531.194,Z 808.710,A 0.000,B 0.000,C 90.000,E1 343.866} C_DIS
LIN {X -0.168,Y -538.748,Z 808.707,A 0.000,B 0.000,C 90.000,E1 343.323} C_DIS
LIN {X 0.325,Y -547.592,Z 808.704,A 0.000,B 0.000,C 90.000,E1 342.598} C_DIS
LIN {X -0.116,Y -557.600,Z 808.699,A 0.000,B 0.000,C 90.000,E1 341.819} C_DIS
LIN {X -0.343,Y -564.317,Z 808.696,A 0.000,B 0.000,C 90.000,E1 341.221} C_DIS
LIN {X 0.151,Y -568.260,Z 808.693,A 0.000,B 0.000,C 90.000,E1 340.786} C_DIS
LIN {X 0.327,Y -573.314,Z 808.690,A 0.000,B 0.000,C 90.000,E1 340.242} C_DIS
LIN {X 0.281,Y -580.144,Z 808.686,A 0.000,B 0.000,C 90.000,E1 339.444} C_DIS
LIN {X -0.148,Y -583.294,Z 808.684,A 0.000,B 0.000,C 90.000,E1 339.082} C_DIS
LIN {X -0.223,Y -589.114,Z 808.679,A 0.000,B 0.000,C 90.000,E1 338.284} C_DIS
LIN {X 0.206,Y -596.276,Z 808.673,A 0.000,B 0.000,C 90.000,E1 337.177} C_DIS
LIN {X -0.054,Y -601.215,Z 808.669,A 0.000,B 0.000,C 90.000,E1 336.410} C_DIS
LIN {X -0.011,Y -607.551,Z 808.663,A 0.000,B 0.000,C 90.000,E1 335.357} C_DIS
LIN {X -0.166,Y -612.906,Z 808.658,A 0.000,B 0.000,C 90.000,E1 334.460} C_DIS
LIN {X 0.284,Y -619.432,Z 808.652,A 0.000,B 0.000,C 90.000,E1 333.256} C_DIS
LIN {X 0.270,Y -624.243,Z 808.647,A 0.000,B 0.000,C 90.000,E1 332.359} C_DIS
LIN {X -0.261,Y -627.479,Z 808.643,A 0.000,B 0.000,C 90.000,E1 331.769} C_DIS
LIN {X 0.158,Y -633.576,Z 808.636,A 0.000,B 0.000,C 90.000,E1 330.461} C_DIS
LIN {X 0.125,Y -639.334,Z 808.629,A 0.000,B 0.000,C 90.000,E1 329.203} C_DIS
LIN {X 0.062,Y -642.639,Z 808.625,A 0.000,B 0.000,C 90.000,E1 328.456} C_DIS
LIN {X 0.099,Y -646.654,Z 808.619,A 0.000,B 0.000,C 90.000,E1 327.454} C_DIS
LIN {X 0.069,Y -651.399,Z 808.612,A 0.000,B 0.000,C 90.000,E1 326.215} C_DIS
LIN {X 0.123,Y -653.984,Z 808.608,A 0.000,B 0.000,C 90.000,E1 325.468} C_DIS
LIN {X 0.120,Y -657.257,Z 808.603,A 0.000,B 0.000,C 90.000,E1 324.482} C_DIS
LIN {X 0.135,Y -658.825,Z 808.600,A 0.000,B 0.000,C 90.000,E1 323.989} C_DIS
LIN {X 0.149,Y -662.435,Z 808.593,A 0.000,B 0.000,C 90.000,E1 322.763} C_DIS
LIN {X -0.275,Y -665.080,Z 808.588,A 0.000,B 0.000,C 90.000,E1 321.823} C_DIS
LIN {X -0.167,Y -668.147,Z 808.581,A 0.000,B 0.000,C 90.000,E1 320.598} C_DIS
LIN {X -0.103,Y -670.931,Z 808.574,A 0.000,B 0.000,C 90.000,E1 319.380} C_DIS
LIN {X 0.013,Y -673.497,Z 808.568,A 0.000,B 0.000,C 90.000,E1 318.162} C_DIS
LIN {X -0.381,Y -674.899,Z 808.564,A 0.000,B 0.000,C 90.000,E1 317.472} C_DIS
LIN {X 0.283,Y -677.478,Z 808.556,A 0.000,B 0.000,C 90.000,E1 315.972} C_DIS
LIN {X -0.047,Y -678.937,Z 808.550,A 0.000,B 0.000,C 90.000,E1 315.040} C_DIS
LIN {X -0.273,Y -680.931,Z 808.542,A 0.000,B 0.000,C 90.000,E1 313.623} C_DIS
LIN {X 0.048,Y -682.714,Z 808.534,A 0.000,B 0.000,C 90.000,E1 312.162} C_DIS
LIN {X -0.158,Y -684.161,Z 808.528,A 0.000,B 0.000,C 90.000,E1 310.987} C_DIS
LIN {X -0.225,Y -685.655,Z 808.520,A 0.000,B 0.000,C 90.000,E1 309.564} C_DIS
LIN {X -0.316,Y -686.828,Z 808.513,A 0.000,B 0.000,C 90.000,E1 308.382} C_DIS
LIN {X -0.222,Y -688.139,Z 808.505,A 0.000,B 0.000,C 90.000,E1 306.950} C_DIS
LIN {X -0.102,Y -689.318,Z 808.497,A 0.000,B 0.000,C 90.000,E1 305.518} C_DIS
LIN {X -0.003,Y -690.239,Z 808.491,A 0.000,B 0.000,C 90.000,E1 304.326} C_DIS
LIN {X -0.041,Y -691.422,Z 808.482,A 0.000,B 0.000,C 90.000,E1 302.673} C_DIS
LIN {X -0.195,Y -692.890,Z 808.471,A 0.000,B 0.000,C 90.000,E1 300.797} C_DIS
LIN {X 0.398,Y -693.834,Z 808.463,A 0.000,B 0.000,C 90.000,E1 299.333} C_DIS
LIN {X 0.232,Y -695.055,Z 808.453,A 0.000,B 0.000,C 90.000,E1 297.462} C_DIS
LIN {X 0.100,Y -696.376,Z 808.442,A 0.000,B 0.000,C 90.000,E1 295.591} C_DIS
LIN {X -0.054,Y -696.951,Z 808.438,A 0.000,B 0.000,C 90.000,E1 294.899} C_DIS
LIN {X -0.201,Y -697.237,Z 808.434,A 0.000,B 0.000,C 90.000,E1 294.207} C_DIS
LIN {X 0.314,Y -696.897,Z 808.432,A 0.000,B 0.000,C 90.000,E1 293.695} C_DIS
LIN {X -0.347,Y -696.428,Z 808.431,A 0.000,B 0.000,C 90.000,E1 293.515} C_DIS
LIN {X -0.113,Y -694.680,Z 808.428,A 0.000,B 0.000,C 90.000,E1 293.025} C_DIS
LIN {X 0.013,Y -694.118,Z 808.427,A 0.000,B 0.000,C 90.000,E1 292.898} C_DIS
LIN {X 0.137,Y -693.259,Z 808.427,A 0.000,B 0.000,C 90.000,E1 292.770} C_DIS
LIN {X 0.258,Y -691.986,Z 808.426,A 0.000,B 0.000,C 90.000,E1 292.642} C_DIS
LIN {X -0.258,Y -689.167,Z 808.425,A 0.000,B 0.000,C 90.000,E1 292.461} C_DIS
LIN {X 0.366,Y -686.179,Z 808.424,A 0.000,B 0.000,C 90.000,E1 292.206} C_DIS
LIN {X -0.169,Y -684.126,Z 808.423,A 0.000,B 0.000,C 90.000,E1 292.153} C_DIS
LIN {X -0.189,Y -682.176,Z 808.423,A 0.000,B 0.000,C 90.000,E1 292.078} C_DIS
LIN {X -0.316,Y -674.543,Z 808.421,A 0.000,B 0.000,C 90.000,E1 291.844} C_DIS
LIN {X -0.120,Y -672.483,Z 808.421,A 0.000,B 0.000,C 90.000,E1 291.770} C_DIS
LIN {X -0.223,Y -661.230,Z 808.420,A 0.000,B 0.000,C 90.000,E1 291.589} C_DIS
LIN {X 0.360,Y -645.349,Z 808.418,A 0.000,B 0.000,C 90.000,E1 291.280} C_DIS
LIN {X 0.107,Y -627.848,Z 808.417,A 0.000,B 0.000,C 90.000,E1 290.972} C_DIS
LIN {X 0.140,Y -614.433,Z 808.415,A 0.000,B 0.000,C 90.000,E1 290.663} C_DIS
LIN {X 0.293,Y -606.434,Z 808.414,A 0.000,B 0.000,C 90.000,E1 290.429} C_DIS
LIN {X -0.237,Y -596.759,Z 808.412,A 0.000,B 0.000,C 90.000,E1 290.120} C_DIS
LIN {X -0.311,Y -595.343,Z 808.411,A 0.000,B 0.000,C 90.000,E1 290.066} C_DIS
LIN {X -0.241,Y -594.220,Z 808.411,A 0.000,B 0.000,C 90.000,E1 289.993} C_DIS
LIN {X 0.259,Y -590.200,Z 808.410,A 0.000,B 0.000,C 90.000,E1 289.758} C_DIS
LIN {X 0.006,Y -589.202,Z 808.410,A 0.000,B 0.000,C 90.000,E1 289.704} C_DIS
LIN {X -0.049,Y -588.489,Z 808.409,A 0.000,B 0.000,C 90.000,E1 289.631} C_DIS
LIN {X -0.112,Y -587.014,Z 808.408,A 0.000,B 0.000,C 90.000,E1 289.504} C_DIS
LIN {X -0.028,Y -586.232,Z 808.408,A 0.000,B 0.000,C 90.000,E1 289.450} C_DIS
LIN {X -0.071,Y -586.190,Z 808.408,A 0.000,B 0.000,C 90.000,E1 289.450} C_DIS
LIN {X 0.114,Y -586.178,Z 808.407,A 0.000,B 0.000,C 90.000,E1 289.214} C_DIS
LIN {X -0.098,Y -587.602,Z 808.405,A 0.000,B 0.000,C 90.000,E1 288.833} C_DIS
LIN {X 0.199,Y -588.165,Z 808.404,A 0.000,B 0.000,C 90.000,E1 288.671} C_DIS
LIN {X -0.085,Y -591.101,Z 808.401,A 0.000,B 0.000,C 90.000,E1 288.181} C_DIS
LIN {X 0.170,Y -597.585,Z 808.395,A 0.000,B 0.000,C 90.000,E1 287.094} C_DIS
LIN {X -0.185,Y -599.619,Z 808.393,A 0.000,B 0.000,C 90.000,E1 286.732} C_DIS
LIN {X 0.102,Y -600.889,Z 808.391,A 0.000,B 0.000,C 90.000,E1 286.441} C_DIS
LIN {X 0.282,Y -603.070,Z 808.389,A 0.000,B 0.000,C 90.000,E1 285.898} C_DIS
LIN {X 0.042,Y -605.757,Z 808.384,A 0.000,B 0.000,C 90.000,E1 285.134} C_DIS
LIN {X 0.251,Y -606.753,Z 808.381,A 0.000,B 0.000,C 90.000,E1 284.592} C_DIS
LIN {X -0.013,Y -607.209,Z 808.380,A 0.000,B 0.000,C 90.000,E1 284.356} C_DIS
LIN {X 0.052,Y -607.816,Z 808.377,A 0.000,B 0.000,C 90.000,E1 283.828} C_DIS
LIN {X 0.125,Y -608.124,Z 808.374,A 0.000,B 0.000,C 90.000,E1 283.300} C_DIS
LIN {X -0.133,Y -608.078,Z 808.373,A 0.000,B 0.000,C 90.000,E1 283.063} C_DIS
LIN {X -0.056,Y -607.571,Z 808.370,A 0.000,B 0.000,C 90.000,E1 282.535} C_DIS
LIN {X 0.018,Y -606.436,Z 808.367,A 0.000,B 0.000,C 90.000,E1 282.007} C_DIS
LIN {X 0.084,Y -605.088,Z 808.364,A 0.000,B 0.000,C 90.000,E1 281.478} C_DIS
LIN {X 0.139,Y -603.229,Z 808.361,A 0.000,B 0.000,C 90.000,E1 280.950} C_DIS
LIN {X 0.071,Y -601.105,Z 808.358,A 0.000,B 0.000,C 90.000,E1 280.433} C_DIS
LIN {X -0.208,Y -599.877,Z 808.357,A 0.000,B 0.000,C 90.000,E1 280.197} C_DIS
LIN {X -0.192,Y -596.835,Z 808.354,A 0.000,B 0.000,C 90.000,E1 279.670} C_DIS
LIN {X -0.298,Y -593.306,Z 808.351,A 0.000,B 0.000,C 90.000,E1 279.151} C_DIS
LIN {X 0.180,Y -592.190,Z 808.350,A 0.000,B 0.000,C 90.000,E1 278.973} C_DIS
LIN {X -0.227,Y -588.243,Z 808.348,A 0.000,B 0.000,C 90.000,E1 278.624} C_DIS
LIN {X 0.220,Y -586.797,Z 808.347,A 0.000,B 0.000,C 90.000,E1 278.454} C_DIS
LIN {X 0.213,Y -583.478,Z 808.346,A 0.000,B 0.000,C 90.000,E1 278.219} C_DIS
LIN {X -0.224,Y -577.882,Z 808.344,A 0.000,B 0.000,C 90.000,E1 277.992} C_DIS
LIN {X 0.215,Y -575.753,Z 808.344,A 0.000,B 0.000,C 90.000,E1 277.871} C_DIS
LIN {X 0.152,Y -569.929,Z 808.343,A 0.000,B 0.000,C 90.000,E1 277.701} C_DIS
LIN {X -0.201,Y -563.104,Z 808.342,A 0.000,B 0.000,C 90.000,E1 277.587} C_DIS
LIN {X -0.028,Y -556.725,Z 808.342,A 0.000,B 0.000,C 90.000,E1 277.530} C_DIS
LIN {X 0.190,Y -553.099,Z 808.341,A 0.000,B 0.000,C 90.000,E1 277.409} C_DIS
LIN {X 0.161,Y -553.081,Z 808.341,A 0.000,B 0.000,C 90.000,E1 277.409} C_DIS
LIN {X -0.181,Y -551.285,Z 808.339,A 0.000,B 0.000,C 90.000,E1 277.068} C_DIS
LIN {X -0.155,Y -550.947,Z 808.339,A 0.000,B 0.000,C 90.000,E1 277.004} C_DIS
LIN {X -0.198,Y -550.929,Z 808.339,A 0.000,B 0.000,C 90.000,E1 277.004} C_DIS
LIN {X -0.246,Y -550.024,Z 808.333,A 0.000,B 0.000,C 90.000,E1 276.024} C_DIS
LIN {X 0.071,Y -549.437,Z 808.326,A 0.000,B 0.000,C 90.000,E1 274.588} C_DIS
LIN {X 0.250,Y -548.960,Z 808.321,A 0.000,B 0.000,C 90.000,E1 273.726} C_DIS
LIN {X -0.029,Y -548.037,Z 808.313,A 0.000,B 0.000,C 90.000,E1 272.350} C_DIS
LIN {X -0.234,Y -546.632,Z 808.302,A 0.000,B 0.000,C 90.000,E1 270.401} C_DIS
LIN {X -0.020,Y -545.696,Z 808.294,A 0.000,B 0.000,C 90.000,E1 268.969} C_DIS
LIN {X -0.197,Y -543.964,Z 808.280,A 0.000,B 0.000,C 90.000,E1 266.445} C_DIS
LIN {X 0.036,Y -542.953,Z 808.271,A 0.000,B 0.000,C 90.000,E1 264.723} C_DIS
LIN {X 0.207,Y -542.144,Z 808.264,A 0.000,B 0.000,C 90.000,E1 263.571} C_DIS
LIN {X -0.106,Y -541.220,Z 808.258,A 0.000,B 0.000,C 90.000,E1 262.470} C_DIS
LIN {X 0.104,Y -540.006,Z 808.250,A 0.000,B 0.000,C 90.000,E1 261.027} C_DIS
LIN {X -0.236,Y -538.968,Z 808.244,A 0.000,B 0.000,C 90.000,E1 259.926} C_DIS
LIN {X 0.226,Y -537.022,Z 808.233,A 0.000,B 0.000,C 90.000,E1 257.881} C_DIS
LIN {X 0.176,Y -535.251,Z 808.223,A 0.000,B 0.000,C 90.000,E1 256.172} C_DIS
LIN {X 0.081,Y -533.300,Z 808.214,A 0.000,B 0.000,C 90.000,E1 254.464} C_DIS
LIN {X 0.229,Y -531.286,Z 808.204,A 0.000,B 0.000,C 90.000,E1 252.725} C_DIS
LIN {X -0.183,Y -529.556,Z 808.196,A 0.000,B 0.000,C 90.000,E1 251.329} C_DIS
LIN {X -0.300,Y -528.125,Z 808.190,A 0.000,B 0.000,C 90.000,E1 250.188} C_DIS
LIN {X -0.093,Y -526.123,Z 808.182,A 0.000,B 0.000,C 90.000,E1 248.720} C_DIS
LIN {X -0.048,Y -523.603,Z 808.172,A 0.000,B 0.000,C 90.000,E1 246.975} C_DIS
LIN {X -0.057,Y -520.977,Z 808.162,A 0.000,B 0.000,C 90.000,E1 245.229} C_DIS
LIN {X 0.134,Y -519.608,Z 808.158,A 0.000,B 0.000,C 90.000,E1 244.332} C_DIS
LIN {X -0.221,Y -516.558,Z 808.148,A 0.000,B 0.000,C 90.000,E1 242.615} C_DIS
LIN {X -0.082,Y -515.016,Z 808.143,A 0.000,B 0.000,C 90.000,E1 241.719} C_DIS
LIN {X -0.163,Y -512.275,Z 808.135,A 0.000,B 0.000,C 90.000,E1 240.255} C_DIS
LIN {X -0.186,Y -510.079,Z 808.128,A 0.000,B 0.000,C 90.000,E1 239.076} C_DIS
LIN {X -0.087,Y -507.057,Z 808.120,A 0.000,B 0.000,C 90.000,E1 237.582} C_DIS
LIN {X -0.044,Y -503.922,Z 808.112,A 0.000,B 0.000,C 90.000,E1 236.087} C_DIS
LIN {X 0.035,Y -502.020,Z 808.107,A 0.000,B 0.000,C 90.000,E1 235.182} C_DIS
LIN {X 0.092,Y -499.998,Z 808.102,A 0.000,B 0.000,C 90.000,E1 234.276} C_DIS
LIN {X 0.160,Y -496.242,Z 808.093,A 0.000,B 0.000,C 90.000,E1 232.763} C_DIS
LIN {X 0.304,Y -493.277,Z 808.087,A 0.000,B 0.000,C 90.000,E1 231.537} C_DIS
LIN {X -0.019,Y -486.029,Z 808.070,A 0.000,B 0.000,C 90.000,E1 228.528} C_DIS
LIN {X 0.235,Y -479.931,Z 808.054,A 0.000,B 0.000,C 90.000,E1 225.729} C_DIS
LIN {X 0.270,Y -475.843,Z 808.044,A 0.000,B 0.000,C 90.000,E1 223.866} C_DIS
LIN {X 0.227,Y -471.753,Z 808.034,A 0.000,B 0.000,C 90.000,E1 222.000} C_DIS
LIN {X -0.217,Y -467.834,Z 808.023,A 0.000,B 0.000,C 90.000,E1 220.172} C_DIS
LIN {X 0.209,Y -464.569,Z 808.014,A 0.000,B 0.000,C 90.000,E1 218.543} C_DIS
LIN {X 0.027,Y -460.593,Z 808.004,A 0.000,B 0.000,C 90.000,E1 216.664} C_DIS
LIN {X 0.224,Y -455.920,Z 807.991,A 0.000,B 0.000,C 90.000,E1 214.405} C_DIS
LIN {X 0.069,Y -452.025,Z 807.981,A 0.000,B 0.000,C 90.000,E1 212.498} C_DIS
LIN {X -0.101,Y -447.405,Z 807.968,A 0.000,B 0.000,C 90.000,E1 210.256} C_DIS
LIN {X 0.019,Y -444.179,Z 807.959,A 0.000,B 0.000,C 90.000,E1 208.615} C_DIS
LIN {X -0.092,Y -440.392,Z 807.948,A 0.000,B 0.000,C 90.000,E1 206.668} C_DIS
LIN {X -0.118,Y -437.283,Z 807.939,A 0.000,B 0.000,C 90.000,E1 205.027} C_DIS
LIN {X 0.024,Y -433.349,Z 807.928,A 0.000,B 0.000,C 90.000,E1 203.025} C_DIS
LIN {X -0.094,Y -429.480,Z 807.917,A 0.000,B 0.000,C 90.000,E1 201.046} C_DIS
LIN {X 0.142,Y -425.013,Z 807.904,A 0.000,B 0.000,C 90.000,E1 198.671} C_DIS
LIN {X 0.153,Y -421.748,Z 807.895,A 0.000,B 0.000,C 90.000,E1 196.985} C_DIS
LIN {X -0.021,Y -418.508,Z 807.885,A 0.000,B 0.000,C 90.000,E1 195.315} C_DIS
LIN {X -0.218,Y -414.567,Z 807.874,A 0.000,B 0.000,C 90.000,E1 193.300} C_DIS
LIN {X 0.193,Y -410.776,Z 807.862,A 0.000,B 0.000,C 90.000,E1 191.186} C_DIS
LIN {X -0.032,Y -406.365,Z 807.849,A 0.000,B 0.000,C 90.000,E1 188.803} C_DIS
LIN {X 0.009,Y -403.737,Z 807.841,A 0.000,B 0.000,C 90.000,E1 187.409} C_DIS
LIN {X -0.103,Y -400.614,Z 807.832,A 0.000,B 0.000,C 90.000,E1 185.682} C_DIS
LIN {X 0.003,Y -396.520,Z 807.818,A 0.000,B 0.000,C 90.000,E1 183.212} C_DIS
LIN {X -0.172,Y -392.212,Z 807.800,A 0.000,B 0.000,C 90.000,E1 180.057} C_DIS
LIN {X 0.055,Y -389.300,Z 807.786,A 0.000,B 0.000,C 90.000,E1 177.535} C_DIS
LIN {X 0.191,Y -388.152,Z 807.780,A 0.000,B 0.000,C 90.000,E1 176.445} C_DIS
LIN {X -0.015,Y -385.410,Z 807.767,A 0.000,B 0.000,C 90.000,E1 173.970} C_DIS
LIN {X -0.177,Y -383.148,Z 807.755,A 0.000,B 0.000,C 90.000,E1 171.837} C_DIS
LIN {X 0.170,Y -381.525,Z 807.745,A 0.000,B 0.000,C 90.000,E1 169.982} C_DIS
LIN {X -0.035,Y -379.046,Z 807.728,A 0.000,B 0.000,C 90.000,E1 167.117} C_DIS
LIN {X -0.039,Y -377.164,Z 807.714,A 0.000,B 0.000,C 90.000,E1 164.574} C_DIS
LIN {X 0.094,Y -375.710,Z 807.698,A 0.000,B 0.000,C 90.000,E1 161.638} C_DIS
LIN {X 0.038,Y -374.988,Z 807.680,A 0.000,B 0.000,C 90.000,E1 158.358} C_DIS
LIN {X -0.173,Y -375.705,Z 807.662,A 0.000,B 0.000,C 90.000,E1 155.101} C_DIS
LIN {X -0.041,Y -376.805,Z 807.651,A 0.000,B 0.000,C 90.000,E1 153.256} C_DIS
LIN {X 0.092,Y -379.266,Z 807.639,A 0.000,B 0.000,C 90.000,E1 151.051} C_DIS
LIN {X 0.038,Y -380.453,Z 807.635,A 0.000,B 0.000,C 90.000,E1 150.333} C_DIS
LIN {X 0.000,Y -382.741,Z 807.629,A 0.000,B 0.000,C 90.000,E1 149.253} C_DIS
LIN {X -0.030,Y -384.664,Z 807.625,A 0.000,B 0.000,C 90.000,E1 148.535} C_DIS
LIN {X 0.155,Y -386.923,Z 807.621,A 0.000,B 0.000,C 90.000,E1 147.788} C_DIS
LIN {X -0.176,Y -389.606,Z 807.617,A 0.000,B 0.000,C 90.000,E1 147.120} C_DIS
LIN {X 0.130,Y -392.437,Z 807.614,A 0.000,B 0.000,C 90.000,E1 146.421} C_DIS
LIN {X -0.048,Y -396.521,Z 807.609,A 0.000,B 0.000,C 90.000,E1 145.642} C_DIS
LIN {X 0.144,Y -398.564,Z 807.607,A 0.000,B 0.000,C 90.000,E1 145.261} C_DIS
LIN {X -0.098,Y -402.035,Z 807.604,A 0.000,B 0.000,C 90.000,E1 144.769} C_DIS
LIN {X 0.017,Y -404.365,Z 807.602,A 0.000,B 0.000,C 90.000,E1 144.402} C_DIS
LIN {X -0.064,Y -409.073,Z 807.599,A 0.000,B 0.000,C 90.000,E1 143.783} C_DIS
LIN {X 0.015,Y -421.359,Z 807.591,A 0.000,B 0.000,C 90.000,E1 142.396} C_DIS
LIN {X -0.046,Y -428.421,Z 807.587,A 0.000,B 0.000,C 90.000,E1 141.618} C_DIS
LIN {X -0.262,Y -432.556,Z 807.584,A 0.000,B 0.000,C 90.000,E1 141.170} C_DIS
LIN {X 0.013,Y -440.522,Z 807.579,A 0.000,B 0.000,C 90.000,E1 140.150} C_DIS
LIN {X -0.043,Y -445.724,Z 807.575,A 0.000,B 0.000,C 90.000,E1 139.504} C_DIS
LIN {X -0.017,Y -451.982,Z 807.571,A 0.000,B 0.000,C 90.000,E1 138.690} C_DIS
LIN {X -0.014,Y -454.624,Z 807.569,A 0.000,B 0.000,C 90.000,E1 138.366} C_DIS
LIN {X 0.058,Y -459.380,Z 807.565,A 0.000,B 0.000,C 90.000,E1 137.715} C_DIS
LIN {X -0.110,Y -466.010,Z 807.560,A 0.000,B 0.000,C 90.000,E1 136.782} C_DIS
LIN {X 0.061,Y -470.881,Z 807.555,A 0.000,B 0.000,C 90.000,E1 135.972} C_DIS
LIN {X -0.234,Y -478.316,Z 807.549,A 0.000,B 0.000,C 90.000,E1 134.757} C_DIS
LIN {X -0.062,Y -481.121,Z 807.546,A 0.000,B 0.000,C 90.000,E1 134.271} C_DIS
LIN {X -0.187,Y -484.833,Z 807.543,A 0.000,B 0.000,C 90.000,E1 133.704} C_DIS
LIN {X 0.095,Y -488.558,Z 807.539,A 0.000,B 0.000,C 90.000,E1 133.056} C_DIS
LIN {X 0.158,Y -492.783,Z 807.535,A 0.000,B 0.000,C 90.000,E1 132.285} C_DIS
LIN {X 0.082,Y -495.241,Z 807.533,A 0.000,B 0.000,C 90.000,E1 131.838} C_DIS
LIN {X -0.104,Y -500.108,Z 807.528,A 0.000,B 0.000,C 90.000,E1 130.987} C_DIS
LIN {X -0.136,Y -502.214,Z 807.525,A 0.000,B 0.000,C 90.000,E1 130.539} C_DIS
LIN {X 0.066,Y -503.550,Z 807.523,A 0.000,B 0.000,C 90.000,E1 130.216} C_DIS
LIN {X 0.040,Y -507.336,Z 807.520,A 0.000,B 0.000,C 90.000,E1 129.519} C_DIS
LIN {X 0.164,Y -510.255,Z 807.516,A 0.000,B 0.000,C 90.000,E1 128.910} C_DIS
LIN {X 0.073,Y -511.461,Z 807.515,A 0.000,B 0.000,C 90.000,E1 128.624} C_DIS
LIN {X 0.056,Y -515.587,Z 807.510,A 0.000,B 0.000,C 90.000,E1 127.810} C_DIS
LIN {X -0.133,Y -521.931,Z 807.502,A 0.000,B 0.000,C 90.000,E1 126.423} C_DIS
LIN {X 0.157,Y -525.636,Z 807.497,A 0.000,B 0.000,C 90.000,E1 125.518} C_DIS
LIN {X 0.087,Y -527.897,Z 807.494,A 0.000,B 0.000,C 90.000,E1 124.945} C_DIS
LIN {X 0.124,Y -532.019,Z 807.488,A 0.000,B 0.000,C 90.000,E1 123.785} C_DIS
LIN {X -0.095,Y -536.477,Z 807.482,A 0.000,B 0.000,C 90.000,E1 122.673} C_DIS
LIN {X 0.066,Y -539.737,Z 807.477,A 0.000,B 0.000,C 90.000,E1 121.799} C_DIS
LIN {X 0.265,Y -542.711,Z 807.472,A 0.000,B 0.000,C 90.000,E1 120.924} C_DIS
LIN {X -0.251,Y -545.461,Z 807.467,A 0.000,B 0.000,C 90.000,E1 120.129} C_DIS
LIN {X -0.264,Y -548.053,Z 807.463,A 0.000,B 0.000,C 90.000,E1 119.283} C_DIS
LIN {X 0.265,Y -551.275,Z 807.456,A 0.000,B 0.000,C 90.000,E1 118.103} C_DIS
LIN {X 0.319,Y -553.402,Z 807.452,A 0.000,B 0.000,C 90.000,E1 117.257} C_DIS
LIN {X 0.144,Y -555.255,Z 807.447,A 0.000,B 0.000,C 90.000,E1 116.437} C_DIS
LIN {X 0.236,Y -556.729,Z 807.442,A 0.000,B 0.000,C 90.000,E1 115.591} C_DIS
LIN {X 0.098,Y -558.024,Z 807.438,A 0.000,B 0.000,C 90.000,E1 114.771} C_DIS
LIN {X 0.067,Y -559.801,Z 807.430,A 0.000,B 0.000,C 90.000,E1 113.387} C_DIS
LIN {X 0.050,Y -561.022,Z 807.424,A 0.000,B 0.000,C 90.000,E1 112.280} C_DIS
LIN {X 0.060,Y -562.108,Z 807.418,A 0.000,B 0.000,C 90.000,E1 111.173} C_DIS
LIN {X 0.082,Y -562.822,Z 807.412,A 0.000,B 0.000,C 90.000,E1 110.066} C_DIS
LIN {X 0.107,Y -563.333,Z 807.405,A 0.000,B 0.000,C 90.000,E1 108.960} C_DIS
LIN {X -0.051,Y -563.680,Z 807.399,A 0.000,B 0.000,C 90.000,E1 107.873} C_DIS
LIN {X 0.093,Y -564.309,Z 807.390,A 0.000,B 0.000,C 90.000,E1 106.205} C_DIS
LIN {X -0.126,Y -565.226,Z 807.379,A 0.000,B 0.000,C 90.000,E1 104.300} C_DIS
LIN {X 0.251,Y -566.625,Z 807.367,A 0.000,B 0.000,C 90.000,E1 102.063} C_DIS
LIN {X -0.299,Y -567.987,Z 807.357,A 0.000,B 0.000,C 90.000,E1 100.197} C_DIS
LIN {X 0.122,Y -569.195,Z 807.347,A 0.000,B 0.000,C 90.000,E1 98.511} C_DIS
LIN {X -0.087,Y -570.320,Z 807.338,A 0.000,B 0.000,C 90.000,E1 96.891} C_DIS
LIN {X 0.223,Y -571.238,Z 807.329,A 0.000,B 0.000,C 90.000,E1 95.220} C_DIS
LIN {X -0.196,Y -571.927,Z 807.322,A 0.000,B 0.000,C 90.000,E1 93.898} C_DIS
LIN {X -0.070,Y -572.519,Z 807.314,A 0.000,B 0.000,C 90.000,E1 92.522} C_DIS
LIN {X -0.222,Y -573.244,Z 807.303,A 0.000,B 0.000,C 90.000,E1 90.630} C_DIS
LIN {X 0.060,Y -573.772,Z 807.294,A 0.000,B 0.000,C 90.000,E1 88.969} C_DIS
LIN {X -0.209,Y -574.178,Z 807.285,A 0.000,B 0.000,C 90.000,E1 87.364} C_DIS
LIN {X -0.044,Y -574.484,Z 807.278,A 0.000,B 0.000,C 90.000,E1 85.988} C_DIS
LIN {X 0.160,Y -574.758,Z 807.270,A 0.000,B 0.000,C 90.000,E1 84.609} C_DIS
LIN {X -0.141,Y -575.071,Z 807.263,A 0.000,B 0.000,C 90.000,E1 83.280} C_DIS
LIN {X 0.097,Y -575.531,Z 807.251,A 0.000,B 0.000,C 90.000,E1 81.084} C_DIS
LIN {X -0.099,Y -575.785,Z 807.243,A 0.000,B 0.000,C 90.000,E1 79.746} C_DIS
LIN {X -0.294,Y -576.081,Z 807.235,A 0.000,B 0.000,C 90.000,E1 78.409} C_DIS
LIN {X -0.036,Y -576.187,Z 807.226,A 0.000,B 0.000,C 90.000,E1 76.756} C_DIS
LIN {X 0.236,Y -576.162,Z 807.220,A 0.000,B 0.000,C 90.000,E1 75.644} C_DIS
LIN {X -0.264,Y -576.070,Z 807.213,A 0.000,B 0.000,C 90.000,E1 74.338} C_DIS
LIN {X -0.051,Y -575.953,Z 807.205,A 0.000,B 0.000,C 90.000,E1 72.960} C_DIS
LIN {X -0.019,Y -575.652,Z 807.196,A 0.000,B 0.000,C 90.000,E1 71.329} C_DIS
LIN {X -0.166,Y -575.114,Z 807.186,A 0.000,B 0.000,C 90.000,E1 69.444} C_DIS
LIN {X 0.033,Y -574.509,Z 807.177,A 0.000,B 0.000,C 90.000,E1 67.794} C_DIS
LIN {X -0.106,Y -573.775,Z 807.168,A 0.000,B 0.000,C 90.000,E1 66.177} C_DIS
LIN {X -0.029,Y -572.860,Z 807.159,A 0.000,B 0.000,C 90.000,E1 64.537} C_DIS
LIN {X -0.070,Y -571.960,Z 807.151,A 0.000,B 0.000,C 90.000,E1 63.179} C_DIS
LIN {X -0.053,Y -571.268,Z 807.146,A 0.000,B 0.000,C 90.000,E1 62.359} C_DIS
LIN {X -0.125,Y -569.874,Z 807.139,A 0.000,B 0.000,C 90.000,E1 61.001} C_DIS
LIN {X 0.229,Y -568.562,Z 807.133,A 0.000,B 0.000,C 90.000,E1 59.871} C_DIS
LIN {X 0.082,Y -567.035,Z 807.127,A 0.000,B 0.000,C 90.000,E1 58.791} C_DIS
LIN {X -0.082,Y -565.247,Z 807.121,A 0.000,B 0.000,C 90.000,E1 57.709} C_DIS
LIN {X -0.068,Y -563.761,Z 807.116,A 0.000,B 0.000,C 90.000,E1 56.882} C_DIS
LIN {X -0.281,Y -561.510,Z 807.110,A 0.000,B 0.000,C 90.000,E1 55.801} C_DIS
LIN {X -0.310,Y -559.612,Z 807.105,A 0.000,B 0.000,C 90.000,E1 54.975} C_DIS
